LIN {X 0,Y 429.867,Z 525.018,A -85,B 0,C 180,E1 -9883.558,E2 -9883.558} C_VEL
LIN {X 0,Y 429.582,Z 537.732,A -85,B 0,C 180,E1 -9884.035,E2 -9884.035} C_VEL
LIN {X 0,Y 429.167,Z 549.996,A -85,B 0,C 180,E1 -9884.689,E2 -9884.689} C_VEL
LIN {X 0,Y 428.602,Z 561.771,A -85,B 0,C 180,E1 -9885.511,E2 -9885.511} C_VEL
LIN {X 0,Y 428.009,Z 572.562,A -85,B 0,C 180,E1 -9886.468,E2 -9886.468} C_VEL
LIN {X 0,Y 427.365,Z 583.19,A -85,B 0,C 180,E1 -9887.656,E2 -9887.656} C_VEL
LIN {X 0,Y 426.826,Z 591.861,A -85,B 0,C 180,E1 -9888.845,E2 -9888.845} C_VEL
LIN {X 0,Y 426.281,Z 598.998,A -85,B 0,C 180,E1 -9890.031,E2 -9890.031} C_VEL
LIN {X 0,Y 425.845,Z 605.937,A -85,B 0,C 180,E1 -9891.458,E2 -9891.458} C_VEL
LIN {X 0,Y 425.404,Z 611.932,A -85,B 0,C 180,E1 -9893.034,E2 -9893.034} C_VEL
LIN {X 0,Y 425.046,Z 615.71,A -85,B 0,C 180,E1 -9894.306,E2 -9894.306} C_VEL
LIN {X 0,Y 425.047,Z 617.92,A -85,B 0,C 180,E1 -9895.258,E2 -9895.258} C_VEL
LIN {X 0,Y 424.825,Z 619.716,A -85,B 0,C 180,E1 -9896.206,E2 -9896.206} C_VEL
LIN {X 0,Y 424.586,Z 621.03,A -85,B 0,C 180,E1 -9897.154,E2 -9897.154} C_VEL
LIN {X 0,Y 424.44,Z 621.926,A -85,B 0,C 180,E1 -9898.102,E2 -9898.102} C_VEL
LIN {X 0,Y 424.38,Z 622.415,A -85,B 0,C 180,E1 -9899.051,E2 -9899.051} C_VEL
LIN {X 0,Y 424.352,Z 622.464,A -85,B 0,C 180,E1 -9900,E2 -9900} C_VEL
LIN {X 0,Y 424.35,Z 622.081,A -85,B 0,C 180,E1 -9900.949,E2 -9900.949} C_VEL
LIN {X 0,Y 424.414,Z 621.294,A -85,B 0,C 180,E1 -9901.898,E2 -9901.898} C_VEL
LIN {X 0,Y 424.575,Z 620.089,A -85,B 0,C 180,E1 -9902.846,E2 -9902.846} C_VEL
LIN {X 0,Y 424.8,Z 617.445,A -85,B 0,C 180,E1 -9904.27,E2 -9904.27} C_VEL
LIN {X 0,Y 424.835,Z 613.78,A -85,B 0,C 180,E1 -9905.696,E2 -9905.696} C_VEL
LIN {X 0,Y 425.13,Z 608.245,A -85,B 0,C 180,E1 -9907.302,E2 -9907.302} C_VEL
LIN {X 0,Y 425.442,Z 601.67,A -85,B 0,C 180,E1 -9908.79,E2 -9908.79} C_VEL
LIN {X 0,Y 425.889,Z 593.769,A -85,B 0,C 180,E1 -9910.218,E2 -9910.218} C_VEL
LIN {X 0,Y 426.316,Z 585.656,A -85,B 0,C 180,E1 -9911.41,E2 -9911.41} C_VEL
LIN {X 0,Y 426.843,Z 575.754,A -85,B 0,C 180,E1 -9912.601,E2 -9912.601} C_VEL
LIN {X 0,Y 427.41,Z 564.895,A -85,B 0,C 180,E1 -9913.66,E2 -9913.66} C_VEL
LIN {X 0,Y 427.808,Z 554.016,A -85,B 0,C 180,E1 -9914.509,E2 -9914.509} C_VEL
LIN {X 0,Y 428.215,Z 541.201,A -85,B 0,C 180,E1 -9915.285,E2 -9915.285} C_VEL
LIN {X 0,Y 428.601,Z 528.47,A -85,B 0,C 180,E1 -9915.85,E2 -9915.85} C_VEL
LIN {X 0,Y 428.82,Z 515.15,A -85,B 0,C 180,E1 -9916.239,E2 -9916.239} C_VEL
LIN {X 0,Y 429.959,Z 434.183,A -85,B 0,C 180,E1 -9917.837,E2 -9917.837} C_VEL
LIN {X 0,Y 425.368,Z 420.644,A -85,B 0,C 180,E1 -9918.296,E2 -9918.296} C_VEL
LIN {X 0,Y 425.296,Z 420.514,A -85,B 0,C 180,E1 -9921.318,E2 -9921.318} C_VEL
LIN {X 0,Y 425.322,Z 420.501,A -85,B 0,C 180,E1 -9924.657,E2 -9924.657} C_VEL
LIN {X 0,Y 425.348,Z 420.498,A -85,B 0,C 180,E1 -9927.558,E2 -9927.558} C_VEL
LIN {X 0,Y 425.291,Z 420.509,A -85,B 0,C 180,E1 -9930.816,E2 -9930.816} C_VEL
LIN {X 0,Y 425.314,Z 420.49,A -85,B 0,C 180,E1 -9934.288,E2 -9934.288} C_VEL
LIN {X 0,Y 425.281,Z 420.51,A -85,B 0,C 180,E1 -9937.694,E2 -9937.694} C_VEL
LIN {X 0,Y 425.282,Z 420.5,A -85,B 0,C 180,E1 -9940.52,E2 -9940.52} C_VEL
LIN {X 0,Y 425.26,Z 420.514,A -85,B 0,C 180,E1 -9943.351,E2 -9943.351} C_VEL
LIN {X 0,Y 425.26,Z 420.506,A -85,B 0,C 180,E1 -9946.649,E2 -9946.649} C_VEL
LIN {X 0,Y 425.288,Z 420.502,A -85,B 0,C 180,E1 -9949.873,E2 -9949.873} C_VEL
LIN {X 0,Y 425.279,Z 420.511,A -85,B 0,C 180,E1 -9952.489,E2 -9952.489} C_VEL
LIN {X 0,Y 425.31,Z 420.505,A -85,B 0,C 180,E1 -9955.817,E2 -9955.817} C_VEL
LIN {X 0,Y 425.293,Z 420.511,A -85,B 0,C 180,E1 -9959.239,E2 -9959.239} C_VEL
LIN {X 0,Y 425.31,Z 420.647,A -85,B 0,C 180,E1 -9962.529,E2 -9962.529} C_VEL
LIN {X 0,Y 428.375,Z 435.146,A -85,B 0,C 180,E1 -9965.269,E2 -9965.269} C_VEL
LIN {X 0,Y 428.559,Z 439.554,A -85,B 0,C 180,E1 -9966.054,E2 -9966.054} C_VEL
LIN {X 0,Y 427.818,Z 458.202,A -85,B 0,C 180,E1 -9969.236,E2 -9969.236} C_VEL
LIN {X 0,Y 427.38,Z 471.342,A -85,B 0,C 180,E1 -9971.337,E2 -9971.337} C_VEL
LIN {X 0,Y 430.685,Z 490.935,A -85,B 0,C 180,E1 -9971.834,E2 -9971.834} C_VEL
LIN {X 0,Y 430.212,Z 535.192,A -85,B 0,C 180,E1 -9972.578,E2 -9972.578} C_VEL
LIN {X 0,Y 429.516,Z 541.034,A -85,B 0,C 180,E1 -9972.65,E2 -9972.65} C_VEL
LIN {X 0,Y 423.913,Z 560.045,A -85,B 0,C 180,E1 -9972.744,E2 -9972.744} C_VEL
LIN {X 0,Y 423.196,Z 565.888,A -85,B 0,C 180,E1 -9972.816,E2 -9972.816} C_VEL
LIN {X 0,Y 422.841,Z 583.643,A -85,B 0,C 180,E1 -9973.152,E2 -9973.152} C_VEL
LIN {X 0,Y 422.427,Z 596.784,A -85,B 0,C 180,E1 -9973.602,E2 -9973.602} C_VEL
LIN {X 0,Y 421.856,Z 609.384,A -85,B 0,C 180,E1 -9974.231,E2 -9974.231} C_VEL
LIN {X 0,Y 421.23,Z 620.994,A -85,B 0,C 180,E1 -9975.012,E2 -9975.012} C_VEL
LIN {X 0,Y 420.569,Z 632.621,A -85,B 0,C 180,E1 -9976.028,E2 -9976.028} C_VEL
LIN {X 0,Y 419.824,Z 643.18,A -85,B 0,C 180,E1 -9977.185,E2 -9977.185} C_VEL
LIN {X 0,Y 419.036,Z 652.058,A -85,B 0,C 180,E1 -9978.389,E2 -9978.389} C_VEL
LIN {X 0,Y 418.455,Z 660.712,A -85,B 0,C 180,E1 -9979.843,E2 -9979.843} C_VEL
LIN {X 0,Y 417.94,Z 667.662,A -85,B 0,C 180,E1 -9981.295,E2 -9981.295} C_VEL
LIN {X 0,Y 417.558,Z 673.185,A -85,B 0,C 180,E1 -9982.748,E2 -9982.748} C_VEL
LIN {X 0,Y 417.394,Z 677.517,A -85,B 0,C 180,E1 -9984.202,E2 -9984.202} C_VEL
LIN {X 0,Y 417.216,Z 679.799,A -85,B 0,C 180,E1 -9985.169,E2 -9985.169} C_VEL
LIN {X 0,Y 417.126,Z 681.659,A -85,B 0,C 180,E1 -9986.136,E2 -9986.136} C_VEL
LIN {X 0,Y 417.137,Z 683.08,A -85,B 0,C 180,E1 -9987.103,E2 -9987.103} C_VEL
LIN {X 0,Y 417.014,Z 684.693,A -85,B 0,C 180,E1 -9989.034,E2 -9989.034} C_VEL
LIN {X 0,Y 417.004,Z 684.929,A -85,B 0,C 180,E1 -9990,E2 -9990} C_VEL
LIN {X 0,Y 417.081,Z 684.152,A -85,B 0,C 180,E1 -9991.931,E2 -9991.931} C_VEL
LIN {X 0,Y 417.137,Z 683.186,A -85,B 0,C 180,E1 -9992.897,E2 -9992.897} C_VEL
LIN {X 0,Y 417.125,Z 681.824,A -85,B 0,C 180,E1 -9993.864,E2 -9993.864} C_VEL
LIN {X 0,Y 417.316,Z 678.955,A -85,B 0,C 180,E1 -9995.315,E2 -9995.315} C_VEL
LIN {X 0,Y 417.48,Z 675.059,A -85,B 0,C 180,E1 -9996.768,E2 -9996.768} C_VEL
LIN {X 0,Y 417.788,Z 670.009,A -85,B 0,C 180,E1 -9998.221,E2 -9998.221} C_VEL
LIN {X 0,Y 418.283,Z 663.641,A -85,B 0,C 180,E1 -9999.673,E2 -9999.673} C_VEL
LIN {X 0,Y 418.866,Z 655.73,A -85,B 0,C 180,E1 -10001.125,E2 -10001.125} C_VEL
LIN {X 0,Y 419.453,Z 647.648,A -85,B 0,C 180,E1 -10002.335,E2 -10002.335} C_VEL
LIN {X 0,Y 420.25,Z 637.715,A -85,B 0,C 180,E1 -10003.54,E2 -10003.54} C_VEL
LIN {X 0,Y 420.88,Z 626.554,A -85,B 0,C 180,E1 -10004.629,E2 -10004.629} C_VEL
LIN {X 0,Y 421.554,Z 615.626,A -85,B 0,C 180,E1 -10005.471,E2 -10005.471} C_VEL
LIN {X 0,Y 422.164,Z 604.555,A -85,B 0,C 180,E1 -10006.129,E2 -10006.129} C_VEL
LIN {X 0,Y 422.695,Z 591.407,A -85,B 0,C 180,E1 -10006.698,E2 -10006.698} C_VEL
LIN {X 0,Y 422.999,Z 579.875,A -85,B 0,C 180,E1 -10007.028,E2 -10007.028} C_VEL
LIN {X 0,Y 423.912,Z 491.011,A -85,B 0,C 180,E1 -10008.562,E2 -10008.562} C_VEL
LIN {X 0,Y 420.501,Z 471.498,A -85,B 0,C 180,E1 -10009.071,E2 -10009.071} C_VEL
LIN {X 0,Y 421.094,Z 454.836,A -85,B 0,C 180,E1 -10011.799,E2 -10011.799} C_VEL
LIN {X 0,Y 421.759,Z 438.57,A -85,B 0,C 180,E1 -10014.62,E2 -10014.62} C_VEL
LIN {X 0,Y 419.397,Z 426.486,A -85,B 0,C 180,E1 -10016.901,E2 -10016.901} C_VEL
LIN {X 0,Y 418.278,Z 421.387,A -85,B 0,C 180,E1 -10017.885,E2 -10017.885} C_VEL
LIN {X 0,Y 418.214,Z 421.393,A -85,B 0,C 180,E1 -10021.396,E2 -10021.396} C_VEL
LIN {X 0,Y 418.268,Z 421.386,A -85,B 0,C 180,E1 -10024.58,E2 -10024.58} C_VEL
LIN {X 0,Y 418.229,Z 421.388,A -85,B 0,C 180,E1 -10027.833,E2 -10027.833} C_VEL
LIN {X 0,Y 418.225,Z 421.386,A -85,B 0,C 180,E1 -10030.948,E2 -10030.948} C_VEL
LIN {X 0,Y 418.212,Z 421.385,A -85,B 0,C 180,E1 -10033.729,E2 -10033.729} C_VEL
LIN {X 0,Y 418.218,Z 421.392,A -85,B 0,C 180,E1 -10036.45,E2 -10036.45} C_VEL
LIN {X 0,Y 418.226,Z 421.387,A -85,B 0,C 180,E1 -10039.13,E2 -10039.13} C_VEL
LIN {X 0,Y 418.231,Z 421.386,A -85,B 0,C 180,E1 -10042.167,E2 -10042.167} C_VEL
LIN {X 0,Y 418.268,Z 421.381,A -85,B 0,C 180,E1 -10045.42,E2 -10045.42} C_VEL
LIN {X 0,Y 418.214,Z 421.394,A -85,B 0,C 180,E1 -10048.604,E2 -10048.604} C_VEL
LIN {X 0,Y 418.259,Z 421.386,A -85,B 0,C 180,E1 -10051.934,E2 -10051.934} C_VEL
LIN {X 0,Y 418.284,Z 421.504,A -85,B 0,C 180,E1 -10052.526,E2 -10052.526} C_VEL
LIN {X 0,Y 421.357,Z 436.857,A -85,B 0,C 180,E1 -10055.355,E2 -10055.355} C_VEL
LIN {X 0,Y 421.519,Z 441.427,A -85,B 0,C 180,E1 -10056.151,E2 -10056.151} C_VEL
LIN {X 0,Y 420.644,Z 462.332,A -85,B 0,C 180,E1 -10059.715,E2 -10059.715} C_VEL
LIN {X 0,Y 420.237,Z 471.969,A -85,B 0,C 180,E1 -10061.346,E2 -10061.346} C_VEL
LIN {X 0,Y 423.175,Z 491.893,A -85,B 0,C 180,E1 -10061.883,E2 -10061.883} C_VEL
LIN {X 0,Y 421.684,Z 582.569,A -85,B 0,C 180,E1 -10063.727,E2 -10063.727} C_VEL
LIN {X 0,Y 421.258,Z 596.208,A -85,B 0,C 180,E1 -10064.208,E2 -10064.208} C_VEL
LIN {X 0,Y 420.744,Z 609.18,A -85,B 0,C 180,E1 -10064.871,E2 -10064.871} C_VEL
LIN {X 0,Y 420.176,Z 621.079,A -85,B 0,C 180,E1 -10065.68,E2 -10065.68} C_VEL
LIN {X 0,Y 419.678,Z 632.631,A -85,B 0,C 180,E1 -10066.688,E2 -10066.688} C_VEL
LIN {X 0,Y 418.978,Z 643.706,A -85,B 0,C 180,E1 -10067.896,E2 -10067.896} C_VEL
LIN {X 0,Y 418.481,Z 652.651,A -85,B 0,C 180,E1 -10069.109,E2 -10069.109} C_VEL
LIN {X 0,Y 418.001,Z 661.355,A -85,B 0,C 180,E1 -10070.565,E2 -10070.565} C_VEL
LIN {X 0,Y 417.597,Z 668.334,A -85,B 0,C 180,E1 -10072.019,E2 -10072.019} C_VEL
LIN {X 0,Y 417.393,Z 673.725,A -85,B 0,C 180,E1 -10073.432,E2 -10073.432} C_VEL
LIN {X 0,Y 417.205,Z 678.792,A -85,B 0,C 180,E1 -10075.168,E2 -10075.168} C_VEL
LIN {X 0,Y 417.098,Z 680.906,A -85,B 0,C 180,E1 -10076.135,E2 -10076.135} C_VEL
LIN {X 0,Y 417.1,Z 682.565,A -85,B 0,C 180,E1 -10077.102,E2 -10077.102} C_VEL
LIN {X 0,Y 417.079,Z 683.807,A -85,B 0,C 180,E1 -10078.069,E2 -10078.069} C_VEL
LIN {X 0,Y 417.014,Z 684.577,A -85,B 0,C 180,E1 -10079.034,E2 -10079.034} C_VEL
LIN {X 0,Y 417.004,Z 684.936,A -85,B 0,C 180,E1 -10080,E2 -10080} C_VEL
LIN {X 0,Y 417.014,Z 684.888,A -85,B 0,C 180,E1 -10080.966,E2 -10080.966} C_VEL
LIN {X 0,Y 417.082,Z 684.371,A -85,B 0,C 180,E1 -10081.931,E2 -10081.931} C_VEL
LIN {X 0,Y 417.168,Z 683.441,A -85,B 0,C 180,E1 -10082.897,E2 -10082.897} C_VEL
LIN {X 0,Y 417.133,Z 682.105,A -85,B 0,C 180,E1 -10083.864,E2 -10083.864} C_VEL
LIN {X 0,Y 417.32,Z 679.213,A -85,B 0,C 180,E1 -10085.315,E2 -10085.315} C_VEL
LIN {X 0,Y 417.472,Z 675.228,A -85,B 0,C 180,E1 -10086.768,E2 -10086.768} C_VEL
LIN {X 0,Y 417.862,Z 669.063,A -85,B 0,C 180,E1 -10088.463,E2 -10088.463} C_VEL
LIN {X 0,Y 418.316,Z 662.293,A -85,B 0,C 180,E1 -10089.916,E2 -10089.916} C_VEL
LIN {X 0,Y 418.97,Z 653.777,A -85,B 0,C 180,E1 -10091.367,E2 -10091.367} C_VEL
LIN {X 0,Y 419.506,Z 645.109,A -85,B 0,C 180,E1 -10092.579,E2 -10092.579} C_VEL
LIN {X 0,Y 420.248,Z 634.771,A -85,B 0,C 180,E1 -10093.747,E2 -10093.747} C_VEL
LIN {X 0,Y 420.895,Z 623.794,A -85,B 0,C 180,E1 -10094.752,E2 -10094.752} C_VEL
LIN {X 0,Y 421.55,Z 612.056,A -85,B 0,C 180,E1 -10095.595,E2 -10095.595} C_VEL
LIN {X 0,Y 422.159,Z 600.099,A -85,B 0,C 180,E1 -10096.254,E2 -10096.254} C_VEL
LIN {X 0,Y 422.622,Z 587.363,A -85,B 0,C 180,E1 -10096.763,E2 -10096.763} C_VEL
LIN {X 0,Y 423.057,Z 571.747,A -85,B 0,C 180,E1 -10097.15,E2 -10097.15} C_VEL
LIN {X 0,Y 424.874,Z 497.19,A -85,B 0,C 180,E1 -10098.803,E2 -10098.803} C_VEL
LIN {X 0,Y 424.848,Z 490.529,A -85,B 0,C 180,E1 -10098.968,E2 -10098.968} C_VEL
LIN {X 0,Y 422.078,Z 475.752,A -85,B 0,C 180,E1 -10099.522,E2 -10099.522} C_VEL
LIN {X 0,Y 421.578,Z 473.354,A -85,B 0,C 180,E1 -10099.635,E2 -10099.635} C_VEL
LIN {X 0,Y 422.554,Z 453.348,A -85,B 0,C 180,E1 -10103.008,E2 -10103.008} C_VEL
LIN {X 0,Y 422.998,Z 441.224,A -85,B 0,C 180,E1 -10105.067,E2 -10105.067} C_VEL
LIN {X 0,Y 421.29,Z 432.304,A -85,B 0,C 180,E1 -10106.771,E2 -10106.771} C_VEL
LIN {X 0,Y 418.268,Z 421.389,A -85,B 0,C 180,E1 -10109.008,E2 -10109.008} C_VEL
LIN {X 0,Y 418.248,Z 421.387,A -85,B 0,C 180,E1 -10112.528,E2 -10112.528} C_VEL
LIN {X 0,Y 418.261,Z 421.385,A -85,B 0,C 180,E1 -10114.841,E2 -10114.841} C_VEL
LIN {X 0,Y 418.257,Z 421.384,A -85,B 0,C 180,E1 -10118.442,E2 -10118.442} C_VEL
LIN {X 0,Y 418.224,Z 421.39,A -85,B 0,C 180,E1 -10120.948,E2 -10120.948} C_VEL
LIN {X 0,Y 418.212,Z 421.391,A -85,B 0,C 180,E1 -10123.729,E2 -10123.729} C_VEL
LIN {X 0,Y 418.212,Z 421.393,A -85,B 0,C 180,E1 -10126.449,E2 -10126.449} C_VEL
LIN {X 0,Y 418.226,Z 421.388,A -85,B 0,C 180,E1 -10129.13,E2 -10129.13} C_VEL
LIN {X 0,Y 418.229,Z 421.388,A -85,B 0,C 180,E1 -10132.167,E2 -10132.167} C_VEL
LIN {X 0,Y 418.267,Z 421.383,A -85,B 0,C 180,E1 -10135.42,E2 -10135.42} C_VEL
LIN {X 0,Y 418.213,Z 421.393,A -85,B 0,C 180,E1 -10138.604,E2 -10138.604} C_VEL
LIN {X 0,Y 418.297,Z 421.512,A -85,B 0,C 180,E1 -10139.671,E2 -10139.671} C_VEL
LIN {X 0,Y 421.825,Z 438.127,A -85,B 0,C 180,E1 -10142.73,E2 -10142.73} C_VEL
LIN {X 0,Y 422.231,Z 441.312,A -85,B 0,C 180,E1 -10143.294,E2 -10143.294} C_VEL
LIN {X 0,Y 421.27,Z 456.799,A -85,B 0,C 180,E1 -10145.875,E2 -10145.875} C_VEL
LIN {X 0,Y 420.182,Z 475.297,A -85,B 0,C 180,E1 -10148.924,E2 -10148.924} C_VEL
LIN {X 0,Y 419.678,Z 485.648,A -85,B 0,C 180,E1 -10150.591,E2 -10150.591} C_VEL
LIN {X 0,Y 421.506,Z 499.502,A -85,B 0,C 180,E1 -10151.079,E2 -10151.079} C_VEL
LIN {X 0,Y 423.449,Z 519.644,A -85,B 0,C 180,E1 -10151.71,E2 -10151.71} C_VEL
LIN {X 0,Y 422.991,Z 539.758,A -85,B 0,C 180,E1 -10152.153,E2 -10152.153} C_VEL
LIN {X 0,Y 422.267,Z 602.397,A -85,B 0,C 180,E1 -10153.222,E2 -10153.222} C_VEL
LIN {X 0,Y 421.922,Z 615.066,A -85,B 0,C 180,E1 -10153.581,E2 -10153.581} C_VEL
LIN {X 0,Y 421.352,Z 627.88,A -85,B 0,C 180,E1 -10154.149,E2 -10154.149} C_VEL
LIN {X 0,Y 420.681,Z 639.693,A -85,B 0,C 180,E1 -10154.868,E2 -10154.868} C_VEL
LIN {X 0,Y 420.07,Z 650.411,A -85,B 0,C 180,E1 -10155.713,E2 -10155.713} C_VEL
LIN {X 0,Y 419.343,Z 661.316,A -85,B 0,C 180,E1 -10156.8,E2 -10156.8} C_VEL
LIN {X 0,Y 418.764,Z 670.173,A -85,B 0,C 180,E1 -10157.89,E2 -10157.89} C_VEL
LIN {X 0,Y 418.228,Z 678.289,A -85,B 0,C 180,E1 -10159.103,E2 -10159.103} C_VEL
LIN {X 0,Y 417.746,Z 686.236,A -85,B 0,C 180,E1 -10160.559,E2 -10160.559} C_VEL
LIN {X 0,Y 417.464,Z 691.604,A -85,B 0,C 180,E1 -10161.773,E2 -10161.773} C_VEL
LIN {X 0,Y 417.236,Z 696.843,A -85,B 0,C 180,E1 -10163.229,E2 -10163.229} C_VEL
LIN {X 0,Y 417.159,Z 700.89,A -85,B 0,C 180,E1 -10164.683,E2 -10164.683} C_VEL
LIN {X 0,Y 417.095,Z 703.869,A -85,B 0,C 180,E1 -10166.135,E2 -10166.135} C_VEL
LIN {X 0,Y 417.116,Z 705.313,A -85,B 0,C 180,E1 -10167.103,E2 -10167.103} C_VEL
LIN {X 0,Y 417.097,Z 706.349,A -85,B 0,C 180,E1 -10168.069,E2 -10168.069} C_VEL
LIN {X 0,Y 417.063,Z 706.954,A -85,B 0,C 180,E1 -10169.034,E2 -10169.034} C_VEL
LIN {X 0,Y 417.066,Z 707.145,A -85,B 0,C 180,E1 -10170,E2 -10170} C_VEL
LIN {X 0,Y 417.063,Z 706.923,A -85,B 0,C 180,E1 -10170.966,E2 -10170.966} C_VEL
LIN {X 0,Y 417.1,Z 706.307,A -85,B 0,C 180,E1 -10171.931,E2 -10171.931} C_VEL
LIN {X 0,Y 417.12,Z 705.298,A -85,B 0,C 180,E1 -10172.897,E2 -10172.897} C_VEL
LIN {X 0,Y 417.103,Z 703.864,A -85,B 0,C 180,E1 -10173.865,E2 -10173.865} C_VEL
LIN {X 0,Y 417.161,Z 700.881,A -85,B 0,C 180,E1 -10175.317,E2 -10175.317} C_VEL
LIN {X 0,Y 417.265,Z 696.83,A -85,B 0,C 180,E1 -10176.771,E2 -10176.771} C_VEL
LIN {X 0,Y 417.523,Z 690.581,A -85,B 0,C 180,E1 -10178.47,E2 -10178.47} C_VEL
LIN {X 0,Y 417.892,Z 683.761,A -85,B 0,C 180,E1 -10179.926,E2 -10179.926} C_VEL
LIN {X 0,Y 418.34,Z 676.779,A -85,B 0,C 180,E1 -10181.139,E2 -10181.139} C_VEL
LIN {X 0,Y 418.915,Z 668.339,A -85,B 0,C 180,E1 -10182.351,E2 -10182.351} C_VEL
LIN {X 0,Y 419.61,Z 657.886,A -85,B 0,C 180,E1 -10183.561,E2 -10183.561} C_VEL
LIN {X 0,Y 420.216,Z 647.518,A -85,B 0,C 180,E1 -10184.529,E2 -10184.529} C_VEL
LIN {X 0,Y 420.91,Z 636.08,A -85,B 0,C 180,E1 -10185.371,E2 -10185.371} C_VEL
LIN {X 0,Y 421.565,Z 624.189,A -85,B 0,C 180,E1 -10186.029,E2 -10186.029} C_VEL
LIN {X 0,Y 422.051,Z 611.321,A -85,B 0,C 180,E1 -10186.538,E2 -10186.538} C_VEL
LIN {X 0,Y 422.393,Z 599.213,A -85,B 0,C 180,E1 -10186.835,E2 -10186.835} C_VEL
LIN {X 0,Y 424.12,Z 518.65,A -85,B 0,C 180,E1 -10188.602,E2 -10188.602} C_VEL
LIN {X 0,Y 421.861,Z 496.233,A -85,B 0,C 180,E1 -10189.288,E2 -10189.288} C_VEL
LIN {X 0,Y 419.734,Z 482.953,A -85,B 0,C 180,E1 -10189.775,E2 -10189.775} C_VEL
LIN {X 0,Y 421.144,Z 461.891,A -85,B 0,C 180,E1 -10193.388,E2 -10193.388} C_VEL
LIN {X 0,Y 422.78,Z 442.084,A -85,B 0,C 180,E1 -10196.935,E2 -10196.935} C_VEL
LIN {X 0,Y 421.389,Z 433.82,A -85,B 0,C 180,E1 -10198.657,E2 -10198.657} C_VEL
LIN {X 0,Y 418.708,Z 423.163,A -85,B 0,C 180,E1 -10201.126,E2 -10201.126} C_VEL
LIN {X 0,Y 418.247,Z 421.391,A -85,B 0,C 180,E1 -10201.605,E2 -10201.605} C_VEL
LIN {X 0,Y 418.261,Z 421.387,A -85,B 0,C 180,E1 -10204.841,E2 -10204.841} C_VEL
LIN {X 0,Y 418.249,Z 421.386,A -85,B 0,C 180,E1 -10208.442,E2 -10208.442} C_VEL
LIN {X 0,Y 418.221,Z 421.39,A -85,B 0,C 180,E1 -10210.948,E2 -10210.948} C_VEL
LIN {X 0,Y 418.211,Z 421.391,A -85,B 0,C 180,E1 -10213.729,E2 -10213.729} C_VEL
LIN {X 0,Y 418.211,Z 421.391,A -85,B 0,C 180,E1 -10216.449,E2 -10216.449} C_VEL
LIN {X 0,Y 418.226,Z 421.392,A -85,B 0,C 180,E1 -10219.13,E2 -10219.13} C_VEL
LIN {X 0,Y 418.231,Z 421.387,A -85,B 0,C 180,E1 -10222.167,E2 -10222.167} C_VEL
LIN {X 0,Y 418.268,Z 421.383,A -85,B 0,C 180,E1 -10225.42,E2 -10225.42} C_VEL
LIN {X 0,Y 418.214,Z 421.392,A -85,B 0,C 180,E1 -10228.604,E2 -10228.604} C_VEL
LIN {X 0,Y 418.294,Z 421.382,A -85,B 0,C 180,E1 -10231.937,E2 -10231.937} C_VEL
LIN {X 0,Y 418.292,Z 421.385,A -85,B 0,C 180,E1 -10235.163,E2 -10235.163} C_VEL
LIN {X 0,Y 418.237,Z 421.392,A -85,B 0,C 180,E1 -10238.304,E2 -10238.304} C_VEL
LIN {X 0,Y 418.286,Z 421.384,A -85,B 0,C 180,E1 -10240.269,E2 -10240.269} C_VEL
LIN {X 0,Y 419.333,Z 424.277,A -85,B 0,C 180,E1 -10240.431,E2 -10240.431} C_VEL
LIN {X 0,Y 424.852,Z 436.499,A -85,B 0,C 180,E1 -10241.141,E2 -10241.141} C_VEL
LIN {X 0,Y 425.474,Z 438.692,A -85,B 0,C 180,E1 -10241.237,E2 -10241.237} C_VEL
LIN {X 0,Y 423.251,Z 524.575,A -85,B 0,C 180,E1 -10243.2,E2 -10243.2} C_VEL
LIN {X 0,Y 422.931,Z 537.536,A -85,B 0,C 180,E1 -10243.684,E2 -10243.684} C_VEL
LIN {X 0,Y 422.527,Z 549.641,A -85,B 0,C 180,E1 -10244.318,E2 -10244.318} C_VEL
LIN {X 0,Y 421.919,Z 562.009,A -85,B 0,C 180,E1 -10245.182,E2 -10245.182} C_VEL
LIN {X 0,Y 421.291,Z 572.639,A -85,B 0,C 180,E1 -10246.125,E2 -10246.125} C_VEL
LIN {X 0,Y 420.681,Z 582.463,A -85,B 0,C 180,E1 -10247.211,E2 -10247.211} C_VEL
LIN {X 0,Y 420.057,Z 591.348,A -85,B 0,C 180,E1 -10248.418,E2 -10248.418} C_VEL
LIN {X 0,Y 419.364,Z 600.004,A -85,B 0,C 180,E1 -10249.865,E2 -10249.865} C_VEL
LIN {X 0,Y 418.892,Z 606.865,A -85,B 0,C 180,E1 -10251.315,E2 -10251.315} C_VEL
LIN {X 0,Y 418.421,Z 612.841,A -85,B 0,C 180,E1 -10252.919,E2 -10252.919} C_VEL
LIN {X 0,Y 418.032,Z 616.579,A -85,B 0,C 180,E1 -10254.211,E2 -10254.211} C_VEL
LIN {X 0,Y 418.026,Z 618.772,A -85,B 0,C 180,E1 -10255.178,E2 -10255.178} C_VEL
LIN {X 0,Y 417.796,Z 620.534,A -85,B 0,C 180,E1 -10256.142,E2 -10256.142} C_VEL
LIN {X 0,Y 417.545,Z 621.824,A -85,B 0,C 180,E1 -10257.106,E2 -10257.106} C_VEL
LIN {X 0,Y 417.387,Z 622.698,A -85,B 0,C 180,E1 -10258.07,E2 -10258.07} C_VEL
LIN {X 0,Y 417.321,Z 623.158,A -85,B 0,C 180,E1 -10259.035,E2 -10259.035} C_VEL
LIN {X 0,Y 417.287,Z 623.161,A -85,B 0,C 180,E1 -10260,E2 -10260} C_VEL
LIN {X 0,Y 417.29,Z 622.749,A -85,B 0,C 180,E1 -10260.965,E2 -10260.965} C_VEL
LIN {X 0,Y 417.362,Z 621.931,A -85,B 0,C 180,E1 -10261.93,E2 -10261.93} C_VEL
LIN {X 0,Y 417.533,Z 620.679,A -85,B 0,C 180,E1 -10262.895,E2 -10262.895} C_VEL
LIN {X 0,Y 417.737,Z 617.983,A -85,B 0,C 180,E1 -10264.342,E2 -10264.342} C_VEL
LIN {X 0,Y 417.775,Z 614.253,A -85,B 0,C 180,E1 -10265.793,E2 -10265.793} C_VEL
LIN {X 0,Y 418.095,Z 608.908,A -85,B 0,C 180,E1 -10267.356,E2 -10267.356} C_VEL
LIN {X 0,Y 418.42,Z 601.988,A -85,B 0,C 180,E1 -10268.938,E2 -10268.938} C_VEL
LIN {X 0,Y 418.881,Z 593.966,A -85,B 0,C 180,E1 -10270.391,E2 -10270.391} C_VEL
LIN {X 0,Y 419.461,Z 583.915,A -85,B 0,C 180,E1 -10271.844,E2 -10271.844} C_VEL
LIN {X 0,Y 420.021,Z 573.444,A -85,B 0,C 180,E1 -10273.055,E2 -10273.055} C_VEL
LIN {X 0,Y 420.609,Z 561.403,A -85,B 0,C 180,E1 -10274.164,E2 -10274.164} C_VEL
LIN {X 0,Y 421.045,Z 549.947,A -85,B 0,C 180,E1 -10274.994,E2 -10274.994} C_VEL
LIN {X 0,Y 421.445,Z 537.954,A -85,B 0,C 180,E1 -10275.661,E2 -10275.661} C_VEL
LIN {X 0,Y 421.816,Z 524.384,A -85,B 0,C 180,E1 -10276.205,E2 -10276.205} C_VEL
LIN {X 0,Y 421.989,Z 509.448,A -85,B 0,C 180,E1 -10276.571,E2 -10276.571} C_VEL
LIN {X 0,Y 423.228,Z 436.539,A -85,B 0,C 180,E1 -10278.039,E2 -10278.039} C_VEL
LIN {X 0,Y 418.339,Z 421.378,A -85,B 0,C 180,E1 -10278.578,E2 -10278.578} C_VEL
LIN {X 0,Y 418.237,Z 421.387,A -85,B 0,C 180,E1 -10281.696,E2 -10281.696} C_VEL
LIN {X 0,Y 418.287,Z 421.379,A -85,B 0,C 180,E1 -10284.864,E2 -10284.864} C_VEL
LIN {X 0,Y 418.292,Z 421.375,A -85,B 0,C 180,E1 -10288.063,E2 -10288.063} C_VEL
LIN {X 0,Y 418.214,Z 421.385,A -85,B 0,C 180,E1 -10291.396,E2 -10291.396} C_VEL
LIN {X 0,Y 418.268,Z 421.368,A -85,B 0,C 180,E1 -10294.58,E2 -10294.58} C_VEL
LIN {X 0,Y 418.23,Z 421.388,A -85,B 0,C 180,E1 -10297.833,E2 -10297.833} C_VEL
LIN {X 0,Y 418.224,Z 421.38,A -85,B 0,C 180,E1 -10300.948,E2 -10300.948} C_VEL
LIN {X 0,Y 418.212,Z 421.39,A -85,B 0,C 180,E1 -10303.729,E2 -10303.729} C_VEL
LIN {X 0,Y 418.211,Z 421.382,A -85,B 0,C 180,E1 -10306.449,E2 -10306.449} C_VEL
LIN {X 0,Y 418.225,Z 421.384,A -85,B 0,C 180,E1 -10309.13,E2 -10309.13} C_VEL
LIN {X 0,Y 418.229,Z 421.39,A -85,B 0,C 180,E1 -10312.167,E2 -10312.167} C_VEL
LIN {X 0,Y 418.268,Z 421.381,A -85,B 0,C 180,E1 -10315.42,E2 -10315.42} C_VEL
LIN {X 0,Y 418.214,Z 421.393,A -85,B 0,C 180,E1 -10318.604,E2 -10318.604} C_VEL
LIN {X 0,Y 418.25,Z 421.393,A -85,B 0,C 180,E1 -10321.934,E2 -10321.934} C_VEL
LIN {X 0,Y 418.249,Z 421.459,A -85,B 0,C 180,E1 -10322.241,E2 -10322.241} C_VEL
LIN {X 0,Y 421.473,Z 436.584,A -85,B 0,C 180,E1 -10325.128,E2 -10325.128} C_VEL
LIN {X 0,Y 421.691,Z 440.869,A -85,B 0,C 180,E1 -10325.9,E2 -10325.9} C_VEL
LIN {X 0,Y 420.88,Z 460.409,A -85,B 0,C 180,E1 -10329.246,E2 -10329.246} C_VEL
LIN {X 0,Y 420.491,Z 471.478,A -85,B 0,C 180,E1 -10331.023,E2 -10331.023} C_VEL
LIN {X 0,Y 423.94,Z 491.511,A -85,B 0,C 180,E1 -10331.543,E2 -10331.543} C_VEL
LIN {X 0,Y 423.196,Z 565.888,A -85,B 0,C 180,E1 -10332.816,E2 -10332.816} C_VEL
LIN {X 0,Y 422.457,Z 571.734,A -85,B 0,C 180,E1 -10332.887,E2 -10332.887} C_VEL
LIN {X 0,Y 419.537,Z 581.213,A -85,B 0,C 180,E1 -10332.955,E2 -10332.955} C_VEL
LIN {X 0,Y 416.566,Z 590.577,A -85,B 0,C 180,E1 -10333.106,E2 -10333.106} C_VEL
LIN {X 0,Y 415.714,Z 596.234,A -85,B 0,C 180,E1 -10333.297,E2 -10333.297} C_VEL
LIN {X 0,Y 415.103,Z 608.488,A -85,B 0,C 180,E1 -10333.904,E2 -10333.904} C_VEL
LIN {X 0,Y 414.482,Z 619.563,A -85,B 0,C 180,E1 -10334.637,E2 -10334.637} C_VEL
LIN {X 0,Y 413.795,Z 630.751,A -85,B 0,C 180,E1 -10335.588,E2 -10335.588} C_VEL
LIN {X 0,Y 413.073,Z 641.318,A -85,B 0,C 180,E1 -10336.721,E2 -10336.721} C_VEL
LIN {X 0,Y 412.258,Z 650.617,A -85,B 0,C 180,E1 -10337.946,E2 -10337.946} C_VEL
LIN {X 0,Y 411.565,Z 659.581,A -85,B 0,C 180,E1 -10339.422,E2 -10339.422} C_VEL
LIN {X 0,Y 410.996,Z 666.773,A -85,B 0,C 180,E1 -10340.899,E2 -10340.899} C_VEL
LIN {X 0,Y 410.514,Z 673.374,A -85,B 0,C 180,E1 -10342.623,E2 -10342.623} C_VEL
LIN {X 0,Y 410.33,Z 677.706,A -85,B 0,C 180,E1 -10344.101,E2 -10344.101} C_VEL
LIN {X 0,Y 410.159,Z 679.988,A -85,B 0,C 180,E1 -10345.085,E2 -10345.085} C_VEL
LIN {X 0,Y 410.039,Z 681.849,A -85,B 0,C 180,E1 -10346.069,E2 -10346.069} C_VEL
LIN {X 0,Y 410.04,Z 683.269,A -85,B 0,C 180,E1 -10347.053,E2 -10347.053} C_VEL
LIN {X 0,Y 410.012,Z 684.265,A -85,B 0,C 180,E1 -10348.035,E2 -10348.035} C_VEL
LIN {X 0,Y 409.927,Z 685.117,A -85,B 0,C 180,E1 -10350,E2 -10350} C_VEL
LIN {X 0,Y 410.012,Z 684.34,A -85,B 0,C 180,E1 -10351.965,E2 -10351.965} C_VEL
LIN {X 0,Y 410.039,Z 683.374,A -85,B 0,C 180,E1 -10352.947,E2 -10352.947} C_VEL
LIN {X 0,Y 410.038,Z 682.012,A -85,B 0,C 180,E1 -10353.931,E2 -10353.931} C_VEL
LIN {X 0,Y 410.262,Z 679.141,A -85,B 0,C 180,E1 -10355.406,E2 -10355.406} C_VEL
LIN {X 0,Y 410.429,Z 675.245,A -85,B 0,C 180,E1 -10356.884,E2 -10356.884} C_VEL
LIN {X 0,Y 410.756,Z 670.194,A -85,B 0,C 180,E1 -10358.362,E2 -10358.362} C_VEL
LIN {X 0,Y 411.276,Z 663.824,A -85,B 0,C 180,E1 -10359.839,E2 -10359.839} C_VEL
LIN {X 0,Y 411.891,Z 655.912,A -85,B 0,C 180,E1 -10361.316,E2 -10361.316} C_VEL
LIN {X 0,Y 412.531,Z 647.826,A -85,B 0,C 180,E1 -10362.545,E2 -10362.545} C_VEL
LIN {X 0,Y 413.342,Z 637.889,A -85,B 0,C 180,E1 -10363.771,E2 -10363.771} C_VEL
LIN {X 0,Y 414.023,Z 626.723,A -85,B 0,C 180,E1 -10364.877,E2 -10364.877} C_VEL
LIN {X 0,Y 414.708,Z 615.788,A -85,B 0,C 180,E1 -10365.733,E2 -10365.733} C_VEL
LIN {X 0,Y 415.357,Z 604.703,A -85,B 0,C 180,E1 -10366.401,E2 -10366.401} C_VEL
LIN {X 0,Y 415.896,Z 591.533,A -85,B 0,C 180,E1 -10366.979,E2 -10366.979} C_VEL
LIN {X 0,Y 416.216,Z 579.958,A -85,B 0,C 180,E1 -10367.314,E2 -10367.314} C_VEL
LIN {X 0,Y 417.218,Z 491.962,A -85,B 0,C 180,E1 -10368.855,E2 -10368.855} C_VEL
LIN {X 0,Y 413.663,Z 471.53,A -85,B 0,C 180,E1 -10369.413,E2 -10369.413} C_VEL
LIN {X 0,Y 414.277,Z 454.824,A -85,B 0,C 180,E1 -10372.177,E2 -10372.177} C_VEL
LIN {X 0,Y 414.903,Z 441.333,A -85,B 0,C 180,E1 -10374.52,E2 -10374.52} C_VEL
LIN {X 0,Y 414.041,Z 435.42,A -85,B 0,C 180,E1 -10375.642,E2 -10375.642} C_VEL
LIN {X 0,Y 411.213,Z 422.265,A -85,B 0,C 180,E1 -10378.208,E2 -10378.208} C_VEL
LIN {X 0,Y 411.185,Z 422.268,A -85,B 0,C 180,E1 -10381.284,E2 -10381.284} C_VEL
LIN {X 0,Y 411.208,Z 422.265,A -85,B 0,C 180,E1 -10384.334,E2 -10384.334} C_VEL
LIN {X 0,Y 411.195,Z 422.264,A -85,B 0,C 180,E1 -10387.974,E2 -10387.974} C_VEL
LIN {X 0,Y 411.166,Z 422.269,A -85,B 0,C 180,E1 -10391.228,E2 -10391.228} C_VEL
LIN {X 0,Y 411.18,Z 422.262,A -85,B 0,C 180,E1 -10394.49,E2 -10394.49} C_VEL
LIN {X 0,Y 411.181,Z 422.259,A -85,B 0,C 180,E1 -10398.195,E2 -10398.195} C_VEL
LIN {X 0,Y 411.222,Z 422.266,A -85,B 0,C 180,E1 -10400.776,E2 -10400.776} C_VEL
LIN {X 0,Y 411.2,Z 422.255,A -85,B 0,C 180,E1 -10404.471,E2 -10404.471} C_VEL
LIN {X 0,Y 411.21,Z 422.265,A -85,B 0,C 180,E1 -10406.873,E2 -10406.873} C_VEL
LIN {X 0,Y 411.213,Z 422.265,A -85,B 0,C 180,E1 -10410.65,E2 -10410.65} C_VEL
LIN {X 0,Y 411.25,Z 422.439,A -85,B 0,C 180,E1 -10412.314,E2 -10412.314} C_VEL
LIN {X 0,Y 414.115,Z 436.278,A -85,B 0,C 180,E1 -10414.895,E2 -10414.895} C_VEL
LIN {X 0,Y 414.64,Z 440.912,A -85,B 0,C 180,E1 -10415.73,E2 -10415.73} C_VEL
LIN {X 0,Y 413.809,Z 459.027,A -85,B 0,C 180,E1 -10418.844,E2 -10418.844} C_VEL
LIN {X 0,Y 413.301,Z 472.115,A -85,B 0,C 180,E1 -10421.086,E2 -10421.086} C_VEL
LIN {X 0,Y 416.298,Z 492.651,A -85,B 0,C 180,E1 -10421.649,E2 -10421.649} C_VEL
LIN {X 0,Y 414.734,Z 583.118,A -85,B 0,C 180,E1 -10423.542,E2 -10423.542} C_VEL
LIN {X 0,Y 414.28,Z 597.317,A -85,B 0,C 180,E1 -10424.061,E2 -10424.061} C_VEL
LIN {X 0,Y 413.747,Z 609.978,A -85,B 0,C 180,E1 -10424.735,E2 -10424.735} C_VEL
LIN {X 0,Y 413.158,Z 622.049,A -85,B 0,C 180,E1 -10425.581,E2 -10425.581} C_VEL
LIN {X 0,Y 412.651,Z 633.194,A -85,B 0,C 180,E1 -10426.582,E2 -10426.582} C_VEL
LIN {X 0,Y 412.033,Z 643.197,A -85,B 0,C 180,E1 -10427.689,E2 -10427.689} C_VEL
LIN {X 0,Y 411.475,Z 652.307,A -85,B 0,C 180,E1 -10428.922,E2 -10428.922} C_VEL
LIN {X 0,Y 410.953,Z 661.109,A -85,B 0,C 180,E1 -10430.401,E2 -10430.401} C_VEL
LIN {X 0,Y 410.543,Z 668.203,A -85,B 0,C 180,E1 -10431.881,E2 -10431.881} C_VEL
LIN {X 0,Y 410.311,Z 674.072,A -85,B 0,C 180,E1 -10433.441,E2 -10433.441} C_VEL
LIN {X 0,Y 410.143,Z 678.802,A -85,B 0,C 180,E1 -10435.085,E2 -10435.085} C_VEL
LIN {X 0,Y 410.013,Z 680.971,A -85,B 0,C 180,E1 -10436.068,E2 -10436.068} C_VEL
LIN {X 0,Y 410,Z 682.657,A -85,B 0,C 180,E1 -10437.052,E2 -10437.052} C_VEL
LIN {X 0,Y 410.008,Z 683.931,A -85,B 0,C 180,E1 -10438.035,E2 -10438.035} C_VEL
LIN {X 0,Y 409.939,Z 684.742,A -85,B 0,C 180,E1 -10439.018,E2 -10439.018} C_VEL
LIN {X 0,Y 409.927,Z 685.124,A -85,B 0,C 180,E1 -10440,E2 -10440} C_VEL
LIN {X 0,Y 409.939,Z 685.101,A -85,B 0,C 180,E1 -10440.982,E2 -10440.982} C_VEL
LIN {X 0,Y 410.013,Z 684.618,A -85,B 0,C 180,E1 -10441.965,E2 -10441.965} C_VEL
LIN {X 0,Y 410.085,Z 683.706,A -85,B 0,C 180,E1 -10442.947,E2 -10442.947} C_VEL
LIN {X 0,Y 410.046,Z 682.393,A -85,B 0,C 180,E1 -10443.931,E2 -10443.931} C_VEL
LIN {X 0,Y 410.274,Z 679.54,A -85,B 0,C 180,E1 -10445.406,E2 -10445.406} C_VEL
LIN {X 0,Y 410.427,Z 675.602,A -85,B 0,C 180,E1 -10446.884,E2 -10446.884} C_VEL
LIN {X 0,Y 410.777,Z 670.448,A -85,B 0,C 180,E1 -10448.362,E2 -10448.362} C_VEL
LIN {X 0,Y 411.252,Z 663.97,A -85,B 0,C 180,E1 -10449.84,E2 -10449.84} C_VEL
LIN {X 0,Y 411.904,Z 655.888,A -85,B 0,C 180,E1 -10451.316,E2 -10451.316} C_VEL
LIN {X 0,Y 412.496,Z 647.57,A -85,B 0,C 180,E1 -10452.546,E2 -10452.546} C_VEL
LIN {X 0,Y 413.254,Z 637.424,A -85,B 0,C 180,E1 -10453.774,E2 -10453.774} C_VEL
LIN {X 0,Y 414.022,Z 625.999,A -85,B 0,C 180,E1 -10454.877,E2 -10454.877} C_VEL
LIN {X 0,Y 414.64,Z 614.851,A -85,B 0,C 180,E1 -10455.735,E2 -10455.735} C_VEL
LIN {X 0,Y 415.342,Z 602.554,A -85,B 0,C 180,E1 -10456.465,E2 -10456.465} C_VEL
LIN {X 0,Y 415.931,Z 589.294,A -85,B 0,C 180,E1 -10457.041,E2 -10457.041} C_VEL
LIN {X 0,Y 416.401,Z 575.022,A -85,B 0,C 180,E1 -10457.433,E2 -10457.433} C_VEL
LIN {X 0,Y 418.435,Z 497.676,A -85,B 0,C 180,E1 -10459.198,E2 -10459.198} C_VEL
LIN {X 0,Y 418.353,Z 490.916,A -85,B 0,C 180,E1 -10459.382,E2 -10459.382} C_VEL
LIN {X 0,Y 415.433,Z 475.804,A -85,B 0,C 180,E1 -10459.99,E2 -10459.99} C_VEL
LIN {X 0,Y 414.951,Z 473.459,A -85,B 0,C 180,E1 -10460.123,E2 -10460.123} C_VEL
LIN {X 0,Y 416.091,Z 452.855,A -85,B 0,C 180,E1 -10463.65,E2 -10463.65} C_VEL
LIN {X 0,Y 416.423,Z 443.697,A -85,B 0,C 180,E1 -10465.223,E2 -10465.223} C_VEL
LIN {X 0,Y 414.75,Z 434.793,A -85,B 0,C 180,E1 -10466.954,E2 -10466.954} C_VEL
LIN {X 0,Y 412.021,Z 424.921,A -85,B 0,C 180,E1 -10469.009,E2 -10469.009} C_VEL
LIN {X 0,Y 411.205,Z 422.27,A -85,B 0,C 180,E1 -10469.598,E2 -10469.598} C_VEL
LIN {X 0,Y 411.209,Z 422.267,A -85,B 0,C 180,E1 -10473.156,E2 -10473.156} C_VEL
LIN {X 0,Y 411.194,Z 422.263,A -85,B 0,C 180,E1 -10476.552,E2 -10476.552} C_VEL
LIN {X 0,Y 411.215,Z 422.261,A -85,B 0,C 180,E1 -10479.728,E2 -10479.728} C_VEL
LIN {X 0,Y 411.176,Z 422.266,A -85,B 0,C 180,E1 -10483.133,E2 -10483.133} C_VEL
LIN {X 0,Y 411.17,Z 422.268,A -85,B 0,C 180,E1 -10485.881,E2 -10485.881} C_VEL
LIN {X 0,Y 411.166,Z 422.267,A -85,B 0,C 180,E1 -10488.772,E2 -10488.772} C_VEL
LIN {X 0,Y 411.206,Z 422.262,A -85,B 0,C 180,E1 -10491.831,E2 -10491.831} C_VEL
LIN {X 0,Y 411.212,Z 422.264,A -85,B 0,C 180,E1 -10495.122,E2 -10495.122} C_VEL
LIN {X 0,Y 411.168,Z 422.267,A -85,B 0,C 180,E1 -10498.003,E2 -10498.003} C_VEL
LIN {X 0,Y 411.246,Z 422.388,A -85,B 0,C 180,E1 -10499.442,E2 -10499.442} C_VEL
LIN {X 0,Y 414.756,Z 438.963,A -85,B 0,C 180,E1 -10502.543,E2 -10502.543} C_VEL
LIN {X 0,Y 415.271,Z 442.084,A -85,B 0,C 180,E1 -10503.109,E2 -10503.109} C_VEL
LIN {X 0,Y 414.293,Z 457.442,A -85,B 0,C 180,E1 -10505.709,E2 -10505.709} C_VEL
LIN {X 0,Y 413.312,Z 474.389,A -85,B 0,C 180,E1 -10508.556,E2 -10508.556} C_VEL
LIN {X 0,Y 412.777,Z 483.043,A -85,B 0,C 180,E1 -10509.997,E2 -10509.997} C_VEL
LIN {X 0,Y 415.029,Z 498.91,A -85,B 0,C 180,E1 -10510.629,E2 -10510.629} C_VEL
LIN {X 0,Y 416.968,Z 520.948,A -85,B 0,C 180,E1 -10511.341,E2 -10511.341} C_VEL
LIN {X 0,Y 416.129,Z 551.917,A -85,B 0,C 180,E1 -10512.064,E2 -10512.064} C_VEL
LIN {X 0,Y 415.459,Z 603.778,A -85,B 0,C 180,E1 -10512.971,E2 -10512.971} C_VEL
LIN {X 0,Y 415.052,Z 616.492,A -85,B 0,C 180,E1 -10513.365,E2 -10513.365} C_VEL
LIN {X 0,Y 414.422,Z 629.964,A -85,B 0,C 180,E1 -10514.004,E2 -10514.004} C_VEL
LIN {X 0,Y 413.722,Z 641.26,A -85,B 0,C 180,E1 -10514.734,E2 -10514.734} C_VEL
LIN {X 0,Y 413.02,Z 652.865,A -85,B 0,C 180,E1 -10515.716,E2 -10515.716} C_VEL
LIN {X 0,Y 412.22,Z 663.27,A -85,B 0,C 180,E1 -10516.819,E2 -10516.819} C_VEL
LIN {X 0,Y 411.704,Z 671.771,A -85,B 0,C 180,E1 -10517.93,E2 -10517.93} C_VEL
LIN {X 0,Y 411.085,Z 679.58,A -85,B 0,C 180,E1 -10519.16,E2 -10519.16} C_VEL
LIN {X 0,Y 410.63,Z 687.184,A -85,B 0,C 180,E1 -10520.642,E2 -10520.642} C_VEL
LIN {X 0,Y 410.3,Z 693.287,A -85,B 0,C 180,E1 -10522.124,E2 -10522.124} C_VEL
LIN {X 0,Y 410.101,Z 698.385,A -85,B 0,C 180,E1 -10523.701,E2 -10523.701} C_VEL
LIN {X 0,Y 410.077,Z 701.787,A -85,B 0,C 180,E1 -10525.084,E2 -10525.084} C_VEL
LIN {X 0,Y 410.008,Z 703.677,A -85,B 0,C 180,E1 -10526.068,E2 -10526.068} C_VEL
LIN {X 0,Y 410.013,Z 705.141,A -85,B 0,C 180,E1 -10527.052,E2 -10527.052} C_VEL
LIN {X 0,Y 410.025,Z 706.178,A -85,B 0,C 180,E1 -10528.035,E2 -10528.035} C_VEL
LIN {X 0,Y 409.985,Z 706.773,A -85,B 0,C 180,E1 -10529.018,E2 -10529.018} C_VEL
LIN {X 0,Y 409.985,Z 706.957,A -85,B 0,C 180,E1 -10530,E2 -10530} C_VEL
LIN {X 0,Y 409.985,Z 706.735,A -85,B 0,C 180,E1 -10530.982,E2 -10530.982} C_VEL
LIN {X 0,Y 410.028,Z 706.118,A -85,B 0,C 180,E1 -10531.965,E2 -10531.965} C_VEL
LIN {X 0,Y 410.018,Z 705.108,A -85,B 0,C 180,E1 -10532.948,E2 -10532.948} C_VEL
LIN {X 0,Y 410.016,Z 703.674,A -85,B 0,C 180,E1 -10533.931,E2 -10533.931} C_VEL
LIN {X 0,Y 410.053,Z 700.691,A -85,B 0,C 180,E1 -10535.409,E2 -10535.409} C_VEL
LIN {X 0,Y 410.19,Z 696.641,A -85,B 0,C 180,E1 -10536.888,E2 -10536.888} C_VEL
LIN {X 0,Y 410.476,Z 690.392,A -85,B 0,C 180,E1 -10538.616,E2 -10538.616} C_VEL
LIN {X 0,Y 410.876,Z 683.574,A -85,B 0,C 180,E1 -10540.098,E2 -10540.098} C_VEL
LIN {X 0,Y 411.325,Z 676.592,A -85,B 0,C 180,E1 -10541.332,E2 -10541.332} C_VEL
LIN {X 0,Y 411.95,Z 668.155,A -85,B 0,C 180,E1 -10542.563,E2 -10542.563} C_VEL
LIN {X 0,Y 412.676,Z 657.704,A -85,B 0,C 180,E1 -10543.794,E2 -10543.794} C_VEL
LIN {X 0,Y 413.321,Z 647.34,A -85,B 0,C 180,E1 -10544.777,E2 -10544.777} C_VEL
LIN {X 0,Y 414.065,Z 635.909,A -85,B 0,C 180,E1 -10545.632,E2 -10545.632} C_VEL
LIN {X 0,Y 414.742,Z 624.027,A -85,B 0,C 180,E1 -10546.3,E2 -10546.3} C_VEL
LIN {X 0,Y 415.263,Z 611.177,A -85,B 0,C 180,E1 -10546.816,E2 -10546.816} C_VEL
LIN {X 0,Y 416.081,Z 582.204,A -85,B 0,C 180,E1 -10547.542,E2 -10547.542} C_VEL
LIN {X 0,Y 417.524,Z 518.947,A -85,B 0,C 180,E1 -10548.981,E2 -10548.981} C_VEL
LIN {X 0,Y 415.375,Z 497.156,A -85,B 0,C 180,E1 -10549.677,E2 -10549.677} C_VEL
LIN {X 0,Y 412.891,Z 481.972,A -85,B 0,C 180,E1 -10550.259,E2 -10550.259} C_VEL
LIN {X 0,Y 414.319,Z 462.695,A -85,B 0,C 180,E1 -10553.653,E2 -10553.653} C_VEL
LIN {X 0,Y 415.884,Z 445.038,A -85,B 0,C 180,E1 -10556.887,E2 -10556.887} C_VEL
LIN {X 0,Y 415.845,Z 442.32,A -85,B 0,C 180,E1 -10557.422,E2 -10557.422} C_VEL
LIN {X 0,Y 413.997,Z 432.936,A -85,B 0,C 180,E1 -10559.492,E2 -10559.492} C_VEL
LIN {X 0,Y 411.217,Z 422.266,A -85,B 0,C 180,E1 -10562.155,E2 -10562.155} C_VEL
LIN {X 0,Y 411.199,Z 422.267,A -85,B 0,C 180,E1 -10565.529,E2 -10565.529} C_VEL
LIN {X 0,Y 411.212,Z 422.266,A -85,B 0,C 180,E1 -10569.225,E2 -10569.225} C_VEL
LIN {X 0,Y 411.179,Z 422.266,A -85,B 0,C 180,E1 -10572.695,E2 -10572.695} C_VEL
LIN {X 0,Y 411.17,Z 422.268,A -85,B 0,C 180,E1 -10575.881,E2 -10575.881} C_VEL
LIN {X 0,Y 411.166,Z 422.269,A -85,B 0,C 180,E1 -10578.772,E2 -10578.772} C_VEL
LIN {X 0,Y 411.208,Z 422.263,A -85,B 0,C 180,E1 -10581.831,E2 -10581.831} C_VEL
LIN {X 0,Y 411.213,Z 422.264,A -85,B 0,C 180,E1 -10585.122,E2 -10585.122} C_VEL
LIN {X 0,Y 411.168,Z 422.268,A -85,B 0,C 180,E1 -10588.003,E2 -10588.003} C_VEL
LIN {X 0,Y 411.22,Z 422.263,A -85,B 0,C 180,E1 -10591.41,E2 -10591.41} C_VEL
LIN {X 0,Y 411.239,Z 422.261,A -85,B 0,C 180,E1 -10593.619,E2 -10593.619} C_VEL
LIN {X 0,Y 411.205,Z 422.268,A -85,B 0,C 180,E1 -10596.853,E2 -10596.853} C_VEL
LIN {X 0,Y 411.237,Z 422.388,A -85,B 0,C 180,E1 -10599.762,E2 -10599.762} C_VEL
LIN {X 0,Y 412.251,Z 425.158,A -85,B 0,C 180,E1 -10599.923,E2 -10599.923} C_VEL
LIN {X 0,Y 417.669,Z 436.444,A -85,B 0,C 180,E1 -10600.636,E2 -10600.636} C_VEL
LIN {X 0,Y 418.998,Z 439.761,A -85,B 0,C 180,E1 -10600.821,E2 -10600.821} C_VEL
LIN {X 0,Y 417.159,Z 502.972,A -85,B 0,C 180,E1 -10602.32,E2 -10602.32} C_VEL
LIN {X 0,Y 416.659,Z 525.707,A -85,B 0,C 180,E1 -10602.863,E2 -10602.863} C_VEL
LIN {X 0,Y 416.331,Z 538.513,A -85,B 0,C 180,E1 -10603.355,E2 -10603.355} C_VEL
LIN {X 0,Y 415.946,Z 549.46,A -85,B 0,C 180,E1 -10603.938,E2 -10603.938} C_VEL
LIN {X 0,Y 415.333,Z 561.386,A -85,B 0,C 180,E1 -10604.767,E2 -10604.767} C_VEL
LIN {X 0,Y 414.596,Z 572.698,A -85,B 0,C 180,E1 -10605.771,E2 -10605.771} C_VEL
LIN {X 0,Y 414.038,Z 581.664,A -85,B 0,C 180,E1 -10606.753,E2 -10606.753} C_VEL
LIN {X 0,Y 413.286,Z 590.9,A -85,B 0,C 180,E1 -10607.976,E2 -10607.976} C_VEL
LIN {X 0,Y 412.629,Z 599.759,A -85,B 0,C 180,E1 -10609.45,E2 -10609.45} C_VEL
LIN {X 0,Y 412.088,Z 605.777,A -85,B 0,C 180,E1 -10610.676,E2 -10610.676} C_VEL
LIN {X 0,Y 411.573,Z 611.633,A -85,B 0,C 180,E1 -10612.148,E2 -10612.148} C_VEL
LIN {X 0,Y 411.096,Z 616.218,A -85,B 0,C 180,E1 -10613.62,E2 -10613.62} C_VEL
LIN {X 0,Y 411.006,Z 619.624,A -85,B 0,C 180,E1 -10615.095,E2 -10615.095} C_VEL
LIN {X 0,Y 410.768,Z 621.348,A -85,B 0,C 180,E1 -10616.076,E2 -10616.076} C_VEL
LIN {X 0,Y 410.506,Z 622.616,A -85,B 0,C 180,E1 -10617.056,E2 -10617.056} C_VEL
LIN {X 0,Y 410.335,Z 623.467,A -85,B 0,C 180,E1 -10618.037,E2 -10618.037} C_VEL
LIN {X 0,Y 410.261,Z 623.893,A -85,B 0,C 180,E1 -10619.018,E2 -10619.018} C_VEL
LIN {X 0,Y 410.225,Z 623.859,A -85,B 0,C 180,E1 -10620,E2 -10620} C_VEL
LIN {X 0,Y 410.231,Z 623.414,A -85,B 0,C 180,E1 -10620.982,E2 -10620.982} C_VEL
LIN {X 0,Y 410.312,Z 622.563,A -85,B 0,C 180,E1 -10621.963,E2 -10621.963} C_VEL
LIN {X 0,Y 410.492,Z 621.255,A -85,B 0,C 180,E1 -10622.944,E2 -10622.944} C_VEL
LIN {X 0,Y 410.679,Z 618.491,A -85,B 0,C 180,E1 -10624.417,E2 -10624.417} C_VEL
LIN {X 0,Y 410.717,Z 614.684,A -85,B 0,C 180,E1 -10625.893,E2 -10625.893} C_VEL
LIN {X 0,Y 411.046,Z 609.583,A -85,B 0,C 180,E1 -10627.397,E2 -10627.397} C_VEL
LIN {X 0,Y 411.316,Z 603.4,A -85,B 0,C 180,E1 -10628.846,E2 -10628.846} C_VEL
LIN {X 0,Y 411.818,Z 595.558,A -85,B 0,C 180,E1 -10630.323,E2 -10630.323} C_VEL
LIN {X 0,Y 412.259,Z 587.532,A -85,B 0,C 180,E1 -10631.555,E2 -10631.555} C_VEL
LIN {X 0,Y 412.89,Z 576.621,A -85,B 0,C 180,E1 -10632.909,E2 -10632.909} C_VEL
LIN {X 0,Y 413.414,Z 566.7,A -85,B 0,C 180,E1 -10633.907,E2 -10633.907} C_VEL
LIN {X 0,Y 413.913,Z 554.593,A -85,B 0,C 180,E1 -10634.881,E2 -10634.881} C_VEL
LIN {X 0,Y 414.357,Z 541.62,A -85,B 0,C 180,E1 -10635.683,E2 -10635.683} C_VEL
LIN {X 0,Y 414.766,Z 528.511,A -85,B 0,C 180,E1 -10636.267,E2 -10636.267} C_VEL
LIN {X 0,Y 414.986,Z 514.753,A -85,B 0,C 180,E1 -10636.669,E2 -10636.669} C_VEL
LIN {X 0,Y 416.388,Z 438.029,A -85,B 0,C 180,E1 -10638.259,E2 -10638.259} C_VEL
LIN {X 0,Y 411.268,Z 422.259,A -85,B 0,C 180,E1 -10638.822,E2 -10638.822} C_VEL
LIN {X 0,Y 411.204,Z 422.26,A -85,B 0,C 180,E1 -10642.641,E2 -10642.641} C_VEL
LIN {X 0,Y 411.236,Z 422.262,A -85,B 0,C 180,E1 -10645.293,E2 -10645.293} C_VEL
LIN {X 0,Y 411.261,Z 422.253,A -85,B 0,C 180,E1 -10647.478,E2 -10647.478} C_VEL
LIN {X 0,Y 411.192,Z 422.266,A -85,B 0,C 180,E1 -10650.848,E2 -10650.848} C_VEL
LIN {X 0,Y 411.208,Z 422.246,A -85,B 0,C 180,E1 -10654.334,E2 -10654.334} C_VEL
LIN {X 0,Y 411.196,Z 422.264,A -85,B 0,C 180,E1 -10657.974,E2 -10657.974} C_VEL
LIN {X 0,Y 411.166,Z 422.262,A -85,B 0,C 180,E1 -10661.228,E2 -10661.228} C_VEL
LIN {X 0,Y 411.178,Z 422.269,A -85,B 0,C 180,E1 -10664.49,E2 -10664.49} C_VEL
LIN {X 0,Y 411.18,Z 422.266,A -85,B 0,C 180,E1 -10668.195,E2 -10668.195} C_VEL
LIN {X 0,Y 411.216,Z 422.26,A -85,B 0,C 180,E1 -10670.775,E2 -10670.775} C_VEL
LIN {X 0,Y 411.2,Z 422.266,A -85,B 0,C 180,E1 -10674.471,E2 -10674.471} C_VEL
LIN {X 0,Y 411.21,Z 422.265,A -85,B 0,C 180,E1 -10676.873,E2 -10676.873} C_VEL
LIN {X 0,Y 411.213,Z 422.271,A -85,B 0,C 180,E1 -10680.65,E2 -10680.65} C_VEL
LIN {X 0,Y 411.21,Z 422.304,A -85,B 0,C 180,E1 -10681.931,E2 -10681.931} C_VEL
LIN {X 0,Y 414.516,Z 437.722,A -85,B 0,C 180,E1 -10684.921,E2 -10684.921} C_VEL
LIN {X 0,Y 414.821,Z 442.218,A -85,B 0,C 180,E1 -10685.742,E2 -10685.742} C_VEL
LIN {X 0,Y 414.038,Z 460.422,A -85,B 0,C 180,E1 -10688.883,E2 -10688.883} C_VEL
LIN {X 0,Y 413.638,Z 471.666,A -85,B 0,C 180,E1 -10690.703,E2 -10690.703} C_VEL
LIN {X 0,Y 417.2,Z 492.638,A -85,B 0,C 180,E1 -10691.253,E2 -10691.253} C_VEL
LIN {X 0,Y 416.215,Z 577.024,A -85,B 0,C 180,E1 -10692.718,E2 -10692.718} C_VEL
LIN {X 0,Y 415.917,Z 589.831,A -85,B 0,C 180,E1 -10693.053,E2 -10693.053} C_VEL
LIN {X 0,Y 415.714,Z 596.234,A -85,B 0,C 180,E1 -10693.297,E2 -10693.297} C_VEL
LIN {X 0,Y 414.859,Z 600.012,A -85,B 0,C 180,E1 -10693.432,E2 -10693.432} C_VEL
LIN {X 0,Y 408.717,Z 611.708,A -85,B 0,C 180,E1 -10693.837,E2 -10693.837} C_VEL
LIN {X 0,Y 407.909,Z 615.296,A -85,B 0,C 180,E1 -10694.051,E2 -10694.051} C_VEL
LIN {X 0,Y 407.255,Z 625.856,A -85,B 0,C 180,E1 -10694.87,E2 -10694.87} C_VEL
LIN {X 0,Y 406.555,Z 637.198,A -85,B 0,C 180,E1 -10695.995,E2 -10695.995} C_VEL
LIN {X 0,Y 405.641,Z 647.329,A -85,B 0,C 180,E1 -10697.238,E2 -10697.238} C_VEL
LIN {X 0,Y 404.906,Z 655.547,A -85,B 0,C 180,E1 -10698.486,E2 -10698.486} C_VEL
LIN {X 0,Y 404.308,Z 663.559,A -85,B 0,C 180,E1 -10699.989,E2 -10699.989} C_VEL
LIN {X 0,Y 403.715,Z 670.009,A -85,B 0,C 180,E1 -10701.491,E2 -10701.491} C_VEL
LIN {X 0,Y 403.366,Z 675.971,A -85,B 0,C 180,E1 -10703.283,E2 -10703.283} C_VEL
LIN {X 0,Y 403.104,Z 680.177,A -85,B 0,C 180,E1 -10704.999,E2 -10704.999} C_VEL
LIN {X 0,Y 402.957,Z 682.038,A -85,B 0,C 180,E1 -10706,E2 -10706} C_VEL
LIN {X 0,Y 402.942,Z 683.459,A -85,B 0,C 180,E1 -10707.001,E2 -10707.001} C_VEL
LIN {X 0,Y 402.925,Z 684.454,A -85,B 0,C 180,E1 -10708.001,E2 -10708.001} C_VEL
LIN {X 0,Y 402.851,Z 685.306,A -85,B 0,C 180,E1 -10710,E2 -10710} C_VEL
LIN {X 0,Y 402.867,Z 685.115,A -85,B 0,C 180,E1 -10711,E2 -10711} C_VEL
LIN {X 0,Y 402.925,Z 684.528,A -85,B 0,C 180,E1 -10711.999,E2 -10711.999} C_VEL
LIN {X 0,Y 402.942,Z 683.563,A -85,B 0,C 180,E1 -10712.999,E2 -10712.999} C_VEL
LIN {X 0,Y 402.956,Z 682.2,A -85,B 0,C 180,E1 -10714,E2 -10714} C_VEL
LIN {X 0,Y 403.188,Z 679.329,A -85,B 0,C 180,E1 -10715.501,E2 -10715.501} C_VEL
LIN {X 0,Y 403.365,Z 675.432,A -85,B 0,C 180,E1 -10717.006,E2 -10717.006} C_VEL
LIN {X 0,Y 403.713,Z 670.38,A -85,B 0,C 180,E1 -10718.509,E2 -10718.509} C_VEL
LIN {X 0,Y 404.244,Z 664.009,A -85,B 0,C 180,E1 -10720.012,E2 -10720.012} C_VEL
LIN {X 0,Y 404.895,Z 656.094,A -85,B 0,C 180,E1 -10721.514,E2 -10721.514} C_VEL
LIN {X 0,Y 405.614,Z 648.005,A -85,B 0,C 180,E1 -10722.763,E2 -10722.763} C_VEL
LIN {X 0,Y 406.44,Z 638.064,A -85,B 0,C 180,E1 -10724.01,E2 -10724.01} C_VEL
LIN {X 0,Y 407.179,Z 626.892,A -85,B 0,C 180,E1 -10725.133,E2 -10725.133} C_VEL
LIN {X 0,Y 407.881,Z 615.95,A -85,B 0,C 180,E1 -10726.003,E2 -10726.003} C_VEL
LIN {X 0,Y 408.558,Z 604.851,A -85,B 0,C 180,E1 -10726.682,E2 -10726.682} C_VEL
LIN {X 0,Y 409.11,Z 591.66,A -85,B 0,C 180,E1 -10727.27,E2 -10727.27} C_VEL
LIN {X 0,Y 409.461,Z 580.042,A -85,B 0,C 180,E1 -10727.609,E2 -10727.609} C_VEL
LIN {X 0,Y 410.537,Z 493.366,A -85,B 0,C 180,E1 -10729.149,E2 -10729.149} C_VEL
LIN {X 0,Y 406.839,Z 471.608,A -85,B 0,C 180,E1 -10729.756,E2 -10729.756} C_VEL
LIN {X 0,Y 407.47,Z 454.796,A -85,B 0,C 180,E1 -10732.567,E2 -10732.567} C_VEL
LIN {X 0,Y 408.066,Z 442.718,A -85,B 0,C 180,E1 -10734.686,E2 -10734.686} C_VEL
LIN {X 0,Y 406.678,Z 434.508,A -85,B 0,C 180,E1 -10736.26,E2 -10736.26} C_VEL
LIN {X 0,Y 404.16,Z 423.142,A -85,B 0,C 180,E1 -10738.497,E2 -10738.497} C_VEL
LIN {X 0,Y 404.142,Z 423.147,A -85,B 0,C 180,E1 -10741.558,E2 -10741.558} C_VEL
LIN {X 0,Y 404.187,Z 423.139,A -85,B 0,C 180,E1 -10745.016,E2 -10745.016} C_VEL
LIN {X 0,Y 404.155,Z 423.142,A -85,B 0,C 180,E1 -10748.757,E2 -10748.757} C_VEL
LIN {X 0,Y 404.126,Z 423.147,A -85,B 0,C 180,E1 -10751.6,E2 -10751.6} C_VEL
LIN {X 0,Y 404.149,Z 423.138,A -85,B 0,C 180,E1 -10754.522,E2 -10754.522} C_VEL
LIN {X 0,Y 404.142,Z 423.139,A -85,B 0,C 180,E1 -10757.296,E2 -10757.296} C_VEL
LIN {X 0,Y 404.171,Z 423.138,A -85,B 0,C 180,E1 -10759.955,E2 -10759.955} C_VEL
LIN {X 0,Y 404.138,Z 423.131,A -85,B 0,C 180,E1 -10763.125,E2 -10763.125} C_VEL
LIN {X 0,Y 404.147,Z 423.141,A -85,B 0,C 180,E1 -10766.188,E2 -10766.188} C_VEL
LIN {X 0,Y 404.146,Z 423.142,A -85,B 0,C 180,E1 -10769.715,E2 -10769.715} C_VEL
LIN {X 0,Y 404.217,Z 423.216,A -85,B 0,C 180,E1 -10772.067,E2 -10772.067} C_VEL
LIN {X 0,Y 407.344,Z 438.759,A -85,B 0,C 180,E1 -10774.994,E2 -10774.994} C_VEL
LIN {X 0,Y 407.672,Z 443.709,A -85,B 0,C 180,E1 -10775.878,E2 -10775.878} C_VEL
LIN {X 0,Y 406.765,Z 463.632,A -85,B 0,C 180,E1 -10779.334,E2 -10779.334} C_VEL
LIN {X 0,Y 406.368,Z 472.212,A -85,B 0,C 180,E1 -10780.816,E2 -10780.816} C_VEL
LIN {X 0,Y 409.438,Z 492.746,A -85,B 0,C 180,E1 -10781.4,E2 -10781.4} C_VEL
LIN {X 0,Y 407.78,Z 583.374,A -85,B 0,C 180,E1 -10783.35,E2 -10783.35} C_VEL
LIN {X 0,Y 407.345,Z 596.798,A -85,B 0,C 180,E1 -10783.847,E2 -10783.847} C_VEL
LIN {X 0,Y 406.861,Z 608.683,A -85,B 0,C 180,E1 -10784.47,E2 -10784.47} C_VEL
LIN {X 0,Y 406.184,Z 621.683,A -85,B 0,C 180,E1 -10785.38,E2 -10785.38} C_VEL
LIN {X 0,Y 405.693,Z 632.465,A -85,B 0,C 180,E1 -10786.347,E2 -10786.347} C_VEL
LIN {X 0,Y 404.992,Z 643.649,A -85,B 0,C 180,E1 -10787.599,E2 -10787.599} C_VEL
LIN {X 0,Y 404.478,Z 651.889,A -85,B 0,C 180,E1 -10788.727,E2 -10788.727} C_VEL
LIN {X 0,Y 403.914,Z 660.824,A -85,B 0,C 180,E1 -10790.233,E2 -10790.233} C_VEL
LIN {X 0,Y 403.48,Z 668.024,A -85,B 0,C 180,E1 -10791.738,E2 -10791.738} C_VEL
LIN {X 0,Y 403.277,Z 672.87,A -85,B 0,C 180,E1 -10792.993,E2 -10792.993} C_VEL
LIN {X 0,Y 403.116,Z 677.533,A -85,B 0,C 180,E1 -10794.497,E2 -10794.497} C_VEL
LIN {X 0,Y 402.932,Z 681.025,A -85,B 0,C 180,E1 -10795.999,E2 -10795.999} C_VEL
LIN {X 0,Y 402.901,Z 682.742,A -85,B 0,C 180,E1 -10797,E2 -10797} C_VEL
LIN {X 0,Y 402.921,Z 684.043,A -85,B 0,C 180,E1 -10798.001,E2 -10798.001} C_VEL
LIN {X 0,Y 402.867,Z 684.904,A -85,B 0,C 180,E1 -10799,E2 -10799} C_VEL
LIN {X 0,Y 402.851,Z 685.311,A -85,B 0,C 180,E1 -10800,E2 -10800} C_VEL
LIN {X 0,Y 402.867,Z 685.313,A -85,B 0,C 180,E1 -10801,E2 -10801} C_VEL
LIN {X 0,Y 402.946,Z 684.875,A -85,B 0,C 180,E1 -10801.999,E2 -10801.999} C_VEL
LIN {X 0,Y 402.99,Z 683.985,A -85,B 0,C 180,E1 -10802.999,E2 -10802.999} C_VEL
LIN {X 0,Y 402.963,Z 682.69,A -85,B 0,C 180,E1 -10804,E2 -10804} C_VEL
LIN {X 0,Y 403.229,Z 679.884,A -85,B 0,C 180,E1 -10805.501,E2 -10805.501} C_VEL
LIN {X 0,Y 403.391,Z 676.009,A -85,B 0,C 180,E1 -10807.005,E2 -10807.005} C_VEL
LIN {X 0,Y 403.777,Z 670.919,A -85,B 0,C 180,E1 -10808.508,E2 -10808.508} C_VEL
LIN {X 0,Y 404.279,Z 664.48,A -85,B 0,C 180,E1 -10810.011,E2 -10810.011} C_VEL
LIN {X 0,Y 404.974,Z 656.451,A -85,B 0,C 180,E1 -10811.512,E2 -10811.512} C_VEL
LIN {X 0,Y 405.599,Z 648.184,A -85,B 0,C 180,E1 -10812.763,E2 -10812.763} C_VEL
LIN {X 0,Y 406.403,Z 638.126,A -85,B 0,C 180,E1 -10814.011,E2 -10814.011} C_VEL
LIN {X 0,Y 407.225,Z 626.92,A -85,B 0,C 180,E1 -10815.131,E2 -10815.131} C_VEL
LIN {X 0,Y 408.04,Z 614.267,A -85,B 0,C 180,E1 -10816.125,E2 -10816.125} C_VEL
LIN {X 0,Y 408.768,Z 601.705,A -85,B 0,C 180,E1 -10816.866,E2 -10816.866} C_VEL
LIN {X 0,Y 409.357,Z 587.966,A -85,B 0,C 180,E1 -10817.452,E2 -10817.452} C_VEL
LIN {X 0,Y 409.87,Z 572.92,A -85,B 0,C 180,E1 -10817.848,E2 -10817.848} C_VEL
LIN {X 0,Y 412.071,Z 498.322,A -85,B 0,C 180,E1 -10819.621,E2 -10819.621} C_VEL
LIN {X 0,Y 412.036,Z 492.32,A -85,B 0,C 180,E1 -10819.786,E2 -10819.786} C_VEL
LIN {X 0,Y 409.316,Z 478.159,A -85,B 0,C 180,E1 -10820.375,E2 -10820.375} C_VEL
LIN {X 0,Y 408.348,Z 473.789,A -85,B 0,C 180,E1 -10820.601,E2 -10820.601} C_VEL
LIN {X 0,Y 409.54,Z 453.896,A -85,B 0,C 180,E1 -10824.052,E2 -10824.052} C_VEL
LIN {X 0,Y 409.887,Z 446.29,A -85,B 0,C 180,E1 -10825.382,E2 -10825.382} C_VEL
LIN {X 0,Y 408.332,Z 437.503,A -85,B 0,C 180,E1 -10827.135,E2 -10827.135} C_VEL
LIN {X 0,Y 405.956,Z 428.731,A -85,B 0,C 180,E1 -10828.996,E2 -10828.996} C_VEL
LIN {X 0,Y 404.146,Z 423.148,A -85,B 0,C 180,E1 -10830.285,E2 -10830.285} C_VEL
LIN {X 0,Y 404.147,Z 423.144,A -85,B 0,C 180,E1 -10833.812,E2 -10833.812} C_VEL
LIN {X 0,Y 404.138,Z 423.143,A -85,B 0,C 180,E1 -10836.875,E2 -10836.875} C_VEL
LIN {X 0,Y 404.149,Z 423.142,A -85,B 0,C 180,E1 -10840.08,E2 -10840.08} C_VEL
LIN {X 0,Y 404.155,Z 423.141,A -85,B 0,C 180,E1 -10843.084,E2 -10843.084} C_VEL
LIN {X 0,Y 404.15,Z 423.143,A -85,B 0,C 180,E1 -10845.926,E2 -10845.926} C_VEL
LIN {X 0,Y 404.121,Z 423.145,A -85,B 0,C 180,E1 -10848.635,E2 -10848.635} C_VEL
LIN {X 0,Y 404.155,Z 423.141,A -85,B 0,C 180,E1 -10851.492,E2 -10851.492} C_VEL
LIN {X 0,Y 404.186,Z 423.138,A -85,B 0,C 180,E1 -10854.984,E2 -10854.984} C_VEL
LIN {X 0,Y 404.144,Z 423.145,A -85,B 0,C 180,E1 -10858.554,E2 -10858.554} C_VEL
LIN {X 0,Y 404.21,Z 423.285,A -85,B 0,C 180,E1 -10859.214,E2 -10859.214} C_VEL
LIN {X 0,Y 407.933,Z 440.866,A -85,B 0,C 180,E1 -10862.557,E2 -10862.557} C_VEL
LIN {X 0,Y 408.206,Z 445.624,A -85,B 0,C 180,E1 -10863.408,E2 -10863.408} C_VEL
LIN {X 0,Y 406.733,Z 467.279,A -85,B 0,C 180,E1 -10867.121,E2 -10867.121} C_VEL
LIN {X 0,Y 405.981,Z 480.611,A -85,B 0,C 180,E1 -10869.349,E2 -10869.349} C_VEL
LIN {X 0,Y 406.85,Z 487.257,A -85,B 0,C 180,E1 -10869.699,E2 -10869.699} C_VEL
LIN {X 0,Y 408.814,Z 501.778,A -85,B 0,C 180,E1 -10870.267,E2 -10870.267} C_VEL
LIN {X 0,Y 410.557,Z 521.143,A -85,B 0,C 180,E1 -10870.922,E2 -10870.922} C_VEL
LIN {X 0,Y 409.279,Z 565.315,A -85,B 0,C 180,E1 -10871.996,E2 -10871.996} C_VEL
LIN {X 0,Y 408.655,Z 604.923,A -85,B 0,C 180,E1 -10872.71,E2 -10872.71} C_VEL
LIN {X 0,Y 408.149,Z 618.606,A -85,B 0,C 180,E1 -10873.172,E2 -10873.172} C_VEL
LIN {X 0,Y 407.539,Z 630.906,A -85,B 0,C 180,E1 -10873.79,E2 -10873.79} C_VEL
LIN {X 0,Y 406.777,Z 642.672,A -85,B 0,C 180,E1 -10874.595,E2 -10874.595} C_VEL
LIN {X 0,Y 405.981,Z 654.472,A -85,B 0,C 180,E1 -10875.641,E2 -10875.641} C_VEL
LIN {X 0,Y 405.228,Z 664.32,A -85,B 0,C 180,E1 -10876.739,E2 -10876.739} C_VEL
LIN {X 0,Y 404.589,Z 673.252,A -85,B 0,C 180,E1 -10877.968,E2 -10877.968} C_VEL
LIN {X 0,Y 403.907,Z 682.111,A -85,B 0,C 180,E1 -10879.473,E2 -10879.473} C_VEL
LIN {X 0,Y 403.482,Z 689.212,A -85,B 0,C 180,E1 -10880.981,E2 -10880.981} C_VEL
LIN {X 0,Y 403.148,Z 694.852,A -85,B 0,C 180,E1 -10882.487,E2 -10882.487} C_VEL
LIN {X 0,Y 402.987,Z 699.268,A -85,B 0,C 180,E1 -10883.994,E2 -10883.994} C_VEL
LIN {X 0,Y 402.924,Z 703.569,A -85,B 0,C 180,E1 -10885.999,E2 -10885.999} C_VEL
LIN {X 0,Y 402.91,Z 705.018,A -85,B 0,C 180,E1 -10887,E2 -10887} C_VEL
LIN {X 0,Y 402.937,Z 706.032,A -85,B 0,C 180,E1 -10888.001,E2 -10888.001} C_VEL
LIN {X 0,Y 402.907,Z 706.768,A -85,B 0,C 180,E1 -10890,E2 -10890} C_VEL
LIN {X 0,Y 402.91,Z 706.546,A -85,B 0,C 180,E1 -10890.999,E2 -10890.999} C_VEL
LIN {X 0,Y 402.939,Z 705.929,A -85,B 0,C 180,E1 -10891.999,E2 -10891.999} C_VEL
LIN {X 0,Y 402.916,Z 704.919,A -85,B 0,C 180,E1 -10893,E2 -10893} C_VEL
LIN {X 0,Y 402.932,Z 703.485,A -85,B 0,C 180,E1 -10894.001,E2 -10894.001} C_VEL
LIN {X 0,Y 402.953,Z 700.501,A -85,B 0,C 180,E1 -10895.505,E2 -10895.505} C_VEL
LIN {X 0,Y 403.108,Z 696.451,A -85,B 0,C 180,E1 -10897.01,E2 -10897.01} C_VEL
LIN {X 0,Y 403.415,Z 690.203,A -85,B 0,C 180,E1 -10898.768,E2 -10898.768} C_VEL
LIN {X 0,Y 403.853,Z 683.386,A -85,B 0,C 180,E1 -10900.275,E2 -10900.275} C_VEL
LIN {X 0,Y 404.338,Z 676.406,A -85,B 0,C 180,E1 -10901.53,E2 -10901.53} C_VEL
LIN {X 0,Y 404.992,Z 667.97,A -85,B 0,C 180,E1 -10902.783,E2 -10902.783} C_VEL
LIN {X 0,Y 405.768,Z 657.049,A -85,B 0,C 180,E1 -10904.085,E2 -10904.085} C_VEL
LIN {X 0,Y 406.564,Z 645.729,A -85,B 0,C 180,E1 -10905.157,E2 -10905.157} C_VEL
LIN {X 0,Y 407.343,Z 633.771,A -85,B 0,C 180,E1 -10906.025,E2 -10906.025} C_VEL
LIN {X 0,Y 408.026,Z 621.296,A -85,B 0,C 180,E1 -10906.704,E2 -10906.704} C_VEL
LIN {X 0,Y 408.566,Z 609.14,A -85,B 0,C 180,E1 -10907.165,E2 -10907.165} C_VEL
LIN {X 0,Y 409.383,Z 584.846,A -85,B 0,C 180,E1 -10907.838,E2 -10907.838} C_VEL
LIN {X 0,Y 411.129,Z 520.581,A -85,B 0,C 180,E1 -10909.338,E2 -10909.338} C_VEL
LIN {X 0,Y 409.061,Z 498.873,A -85,B 0,C 180,E1 -10910.058,E2 -10910.058} C_VEL
LIN {X 0,Y 406.157,Z 480.875,A -85,B 0,C 180,E1 -10910.789,E2 -10910.789} C_VEL
LIN {X 0,Y 407.577,Z 462.612,A -85,B 0,C 180,E1 -10914.093,E2 -10914.093} C_VEL
LIN {X 0,Y 409.126,Z 446.753,A -85,B 0,C 180,E1 -10917.079,E2 -10917.079} C_VEL
LIN {X 0,Y 409.08,Z 444.01,A -85,B 0,C 180,E1 -10917.637,E2 -10917.637} C_VEL
LIN {X 0,Y 407.243,Z 434.804,A -85,B 0,C 180,E1 -10919.746,E2 -10919.746} C_VEL
LIN {X 0,Y 404.861,Z 425.771,A -85,B 0,C 180,E1 -10922.054,E2 -10922.054} C_VEL
LIN {X 0,Y 404.179,Z 423.141,A -85,B 0,C 180,E1 -10922.818,E2 -10922.818} C_VEL
LIN {X 0,Y 404.143,Z 423.144,A -85,B 0,C 180,E1 -10926.246,E2 -10926.246} C_VEL
LIN {X 0,Y 404.152,Z 423.142,A -85,B 0,C 180,E1 -10928.757,E2 -10928.757} C_VEL
LIN {X 0,Y 404.121,Z 423.148,A -85,B 0,C 180,E1 -10931.599,E2 -10931.599} C_VEL
LIN {X 0,Y 404.147,Z 423.143,A -85,B 0,C 180,E1 -10934.522,E2 -10934.522} C_VEL
LIN {X 0,Y 404.139,Z 423.147,A -85,B 0,C 180,E1 -10937.296,E2 -10937.296} C_VEL
LIN {X 0,Y 404.171,Z 423.139,A -85,B 0,C 180,E1 -10939.955,E2 -10939.955} C_VEL
LIN {X 0,Y 404.139,Z 423.143,A -85,B 0,C 180,E1 -10943.125,E2 -10943.125} C_VEL
LIN {X 0,Y 404.147,Z 423.141,A -85,B 0,C 180,E1 -10946.188,E2 -10946.188} C_VEL
LIN {X 0,Y 404.148,Z 423.143,A -85,B 0,C 180,E1 -10949.715,E2 -10949.715} C_VEL
LIN {X 0,Y 404.197,Z 423.141,A -85,B 0,C 180,E1 -10953.123,E2 -10953.123} C_VEL
LIN {X 0,Y 404.179,Z 423.144,A -85,B 0,C 180,E1 -10955.334,E2 -10955.334} C_VEL
LIN {X 0,Y 404.141,Z 423.147,A -85,B 0,C 180,E1 -10958.581,E2 -10958.581} C_VEL
LIN {X 0,Y 404.178,Z 423.142,A -85,B 0,C 180,E1 -10959.193,E2 -10959.193} C_VEL
LIN {X 0,Y 405.26,Z 426.125,A -85,B 0,C 180,E1 -10959.379,E2 -10959.379} C_VEL
LIN {X 0,Y 410.751,Z 437.204,A -85,B 0,C 180,E1 -10960.149,E2 -10960.149} C_VEL
LIN {X 0,Y 412.677,Z 442.169,A -85,B 0,C 180,E1 -10960.434,E2 -10960.434} C_VEL
LIN {X 0,Y 410.134,Z 525.904,A -85,B 0,C 180,E1 -10962.485,E2 -10962.485} C_VEL
LIN {X 0,Y 409.741,Z 538.83,A -85,B 0,C 180,E1 -10962.983,E2 -10962.983} C_VEL
LIN {X 0,Y 409.288,Z 551.411,A -85,B 0,C 180,E1 -10963.669,E2 -10963.669} C_VEL
LIN {X 0,Y 408.595,Z 563.569,A -85,B 0,C 180,E1 -10964.552,E2 -10964.552} C_VEL
LIN {X 0,Y 407.862,Z 574.235,A -85,B 0,C 180,E1 -10965.531,E2 -10965.531} C_VEL
LIN {X 0,Y 407.25,Z 583.04,A -85,B 0,C 180,E1 -10966.528,E2 -10966.528} C_VEL
LIN {X 0,Y 406.464,Z 592.096,A -85,B 0,C 180,E1 -10967.772,E2 -10967.772} C_VEL
LIN {X 0,Y 405.734,Z 600.86,A -85,B 0,C 180,E1 -10969.268,E2 -10969.268} C_VEL
LIN {X 0,Y 405.155,Z 606.831,A -85,B 0,C 180,E1 -10970.515,E2 -10970.515} C_VEL
LIN {X 0,Y 404.612,Z 612.641,A -85,B 0,C 180,E1 -10972.012,E2 -10972.012} C_VEL
LIN {X 0,Y 404.116,Z 617.176,A -85,B 0,C 180,E1 -10973.509,E2 -10973.509} C_VEL
LIN {X 0,Y 403.988,Z 620.532,A -85,B 0,C 180,E1 -10975.01,E2 -10975.01} C_VEL
LIN {X 0,Y 403.742,Z 622.197,A -85,B 0,C 180,E1 -10976.007,E2 -10976.007} C_VEL
LIN {X 0,Y 403.468,Z 623.431,A -85,B 0,C 180,E1 -10977.005,E2 -10977.005} C_VEL
LIN {X 0,Y 403.286,Z 624.25,A -85,B 0,C 180,E1 -10978.003,E2 -10978.003} C_VEL
LIN {X 0,Y 403.202,Z 624.625,A -85,B 0,C 180,E1 -10979.001,E2 -10979.001} C_VEL
LIN {X 0,Y 403.165,Z 624.553,A -85,B 0,C 180,E1 -10980,E2 -10980} C_VEL
LIN {X 0,Y 403.174,Z 624.077,A -85,B 0,C 180,E1 -10980.999,E2 -10980.999} C_VEL
LIN {X 0,Y 403.264,Z 623.189,A -85,B 0,C 180,E1 -10981.998,E2 -10981.998} C_VEL
LIN {X 0,Y 403.451,Z 621.828,A -85,B 0,C 180,E1 -10982.996,E2 -10982.996} C_VEL
LIN {X 0,Y 403.626,Z 618.997,A -85,B 0,C 180,E1 -10984.494,E2 -10984.494} C_VEL
LIN {X 0,Y 403.667,Z 615.112,A -85,B 0,C 180,E1 -10985.996,E2 -10985.996} C_VEL
LIN {X 0,Y 404.033,Z 609.237,A -85,B 0,C 180,E1 -10987.706,E2 -10987.706} C_VEL
LIN {X 0,Y 404.371,Z 602.447,A -85,B 0,C 180,E1 -10989.251,E2 -10989.251} C_VEL
LIN {X 0,Y 404.892,Z 594.133,A -85,B 0,C 180,E1 -10990.754,E2 -10990.754} C_VEL
LIN {X 0,Y 405.369,Z 585.649,A -85,B 0,C 180,E1 -10992.008,E2 -10992.008} C_VEL
LIN {X 0,Y 406.019,Z 575.275,A -85,B 0,C 180,E1 -10993.259,E2 -10993.259} C_VEL
LIN {X 0,Y 406.623,Z 563.492,A -85,B 0,C 180,E1 -10994.391,E2 -10994.391} C_VEL
LIN {X 0,Y 407.059,Z 552.07,A -85,B 0,C 180,E1 -10995.266,E2 -10995.266} C_VEL
LIN {X 0,Y 407.525,Z 539.12,A -85,B 0,C 180,E1 -10996.018,E2 -10996.018} C_VEL
LIN {X 0,Y 407.927,Z 525.632,A -85,B 0,C 180,E1 -10996.58,E2 -10996.58} C_VEL
LIN {X 0,Y 408.114,Z 510.977,A -85,B 0,C 180,E1 -10996.958,E2 -10996.958} C_VEL
LIN {X 0,Y 409.341,Z 438.527,A -85,B 0,C 180,E1 -10998.503,E2 -10998.503} C_VEL
LIN {X 0,Y 404.204,Z 423.171,A -85,B 0,C 180,E1 -10999.054,E2 -10999.054} C_VEL
LIN {X 0,Y 404.153,Z 423.139,A -85,B 0,C 180,E1 -11002.832,E2 -11002.832} C_VEL
LIN {X 0,Y 404.183,Z 423.137,A -85,B 0,C 180,E1 -11005.767,E2 -11005.767} C_VEL
LIN {X 0,Y 404.197,Z 423.131,A -85,B 0,C 180,E1 -11008,E2 -11008} C_VEL
LIN {X 0,Y 404.142,Z 423.136,A -85,B 0,C 180,E1 -11011.558,E2 -11011.558} C_VEL
LIN {X 0,Y 404.187,Z 423.126,A -85,B 0,C 180,E1 -11015.016,E2 -11015.016} C_VEL
LIN {X 0,Y 404.155,Z 423.141,A -85,B 0,C 180,E1 -11018.757,E2 -11018.757} C_VEL
LIN {X 0,Y 404.126,Z 423.143,A -85,B 0,C 180,E1 -11021.6,E2 -11021.6} C_VEL
LIN {X 0,Y 404.148,Z 423.143,A -85,B 0,C 180,E1 -11024.522,E2 -11024.522} C_VEL
LIN {X 0,Y 404.139,Z 423.143,A -85,B 0,C 180,E1 -11027.296,E2 -11027.296} C_VEL
LIN {X 0,Y 404.171,Z 423.132,A -85,B 0,C 180,E1 -11029.955,E2 -11029.955} C_VEL
LIN {X 0,Y 404.138,Z 423.139,A -85,B 0,C 180,E1 -11033.125,E2 -11033.125} C_VEL
LIN {X 0,Y 404.147,Z 423.14,A -85,B 0,C 180,E1 -11036.188,E2 -11036.188} C_VEL
LIN {X 0,Y 404.146,Z 423.146,A -85,B 0,C 180,E1 -11039.715,E2 -11039.715} C_VEL
LIN {X 0,Y 404.201,Z 423.329,A -85,B 0,C 180,E1 -11041.647,E2 -11041.647} C_VEL
LIN {X 0,Y 407.608,Z 439.051,A -85,B 0,C 180,E1 -11044.739,E2 -11044.739} C_VEL
LIN {X 0,Y 408.034,Z 442.053,A -85,B 0,C 180,E1 -11045.311,E2 -11045.311} C_VEL
LIN {X 0,Y 407.211,Z 460.291,A -85,B 0,C 180,E1 -11048.485,E2 -11048.485} C_VEL
LIN {X 0,Y 406.773,Z 471.756,A -85,B 0,C 180,E1 -11050.364,E2 -11050.364} C_VEL
LIN {X 0,Y 410.491,Z 493.66,A -85,B 0,C 180,E1 -11050.951,E2 -11050.951} C_VEL
LIN {X 0,Y 409.464,Z 577.129,A -85,B 0,C 180,E1 -11052.423,E2 -11052.423} C_VEL
LIN {X 0,Y 409.153,Z 589.98,A -85,B 0,C 180,E1 -11052.764,E2 -11052.764} C_VEL
LIN {X 0,Y 408.579,Z 603.015,A -85,B 0,C 180,E1 -11053.319,E2 -11053.319} C_VEL
LIN {X 0,Y 407.909,Z 615.296,A -85,B 0,C 180,E1 -11054.051,E2 -11054.051} C_VEL
LIN {X 0,Y 407.019,Z 620.56,A -85,B 0,C 180,E1 -11054.41,E2 -11054.41} C_VEL
LIN {X 0,Y 403.762,Z 628.885,A -85,B 0,C 180,E1 -11055.01,E2 -11055.01} C_VEL
LIN {X 0,Y 400.392,Z 636.825,A -85,B 0,C 180,E1 -11055.71,E2 -11055.71} C_VEL
LIN {X 0,Y 399.333,Z 641.398,A -85,B 0,C 180,E1 -11056.22,E2 -11056.22} C_VEL
LIN {X 0,Y 398.388,Z 650.989,A -85,B 0,C 180,E1 -11057.52,E2 -11057.52} C_VEL
LIN {X 0,Y 397.728,Z 658.622,A -85,B 0,C 180,E1 -11058.792,E2 -11058.792} C_VEL
LIN {X 0,Y 397.091,Z 666.061,A -85,B 0,C 180,E1 -11060.32,E2 -11060.32} C_VEL
LIN {X 0,Y 396.534,Z 672.032,A -85,B 0,C 180,E1 -11061.849,E2 -11061.849} C_VEL
LIN {X 0,Y 396.29,Z 676.486,A -85,B 0,C 180,E1 -11063.283,E2 -11063.283} C_VEL
LIN {X 0,Y 396.049,Z 680.365,A -85,B 0,C 180,E1 -11064.91,E2 -11064.91} C_VEL
LIN {X 0,Y 395.88,Z 682.227,A -85,B 0,C 180,E1 -11065.928,E2 -11065.928} C_VEL
LIN {X 0,Y 395.846,Z 683.648,A -85,B 0,C 180,E1 -11066.947,E2 -11066.947} C_VEL
LIN {X 0,Y 395.841,Z 684.643,A -85,B 0,C 180,E1 -11067.965,E2 -11067.965} C_VEL
LIN {X 0,Y 395.779,Z 685.494,A -85,B 0,C 180,E1 -11070,E2 -11070} C_VEL
LIN {X 0,Y 395.796,Z 685.303,A -85,B 0,C 180,E1 -11071.017,E2 -11071.017} C_VEL
LIN {X 0,Y 395.842,Z 684.717,A -85,B 0,C 180,E1 -11072.035,E2 -11072.035} C_VEL
LIN {X 0,Y 395.845,Z 683.751,A -85,B 0,C 180,E1 -11073.053,E2 -11073.053} C_VEL
LIN {X 0,Y 395.879,Z 682.388,A -85,B 0,C 180,E1 -11074.072,E2 -11074.072} C_VEL
LIN {X 0,Y 396.119,Z 679.516,A -85,B 0,C 180,E1 -11075.6,E2 -11075.6} C_VEL
LIN {X 0,Y 396.308,Z 675.618,A -85,B 0,C 180,E1 -11077.131,E2 -11077.131} C_VEL
LIN {X 0,Y 396.684,Z 670.565,A -85,B 0,C 180,E1 -11078.661,E2 -11078.661} C_VEL
LIN {X 0,Y 397.245,Z 664.192,A -85,B 0,C 180,E1 -11080.19,E2 -11080.19} C_VEL
LIN {X 0,Y 397.929,Z 656.276,A -85,B 0,C 180,E1 -11081.719,E2 -11081.719} C_VEL
LIN {X 0,Y 398.703,Z 648.183,A -85,B 0,C 180,E1 -11082.988,E2 -11082.988} C_VEL
LIN {X 0,Y 399.544,Z 638.238,A -85,B 0,C 180,E1 -11084.256,E2 -11084.256} C_VEL
LIN {X 0,Y 400.328,Z 627.061,A -85,B 0,C 180,E1 -11085.398,E2 -11085.398} C_VEL
LIN {X 0,Y 401.072,Z 616.111,A -85,B 0,C 180,E1 -11086.282,E2 -11086.282} C_VEL
LIN {X 0,Y 401.79,Z 604.999,A -85,B 0,C 180,E1 -11086.971,E2 -11086.971} C_VEL
LIN {X 0,Y 402.356,Z 591.787,A -85,B 0,C 180,E1 -11087.569,E2 -11087.569} C_VEL
LIN {X 0,Y 402.719,Z 580.126,A -85,B 0,C 180,E1 -11087.914,E2 -11087.914} C_VEL
LIN {X 0,Y 403.718,Z 493.223,A -85,B 0,C 180,E1 -11089.489,E2 -11089.489} C_VEL
LIN {X 0,Y 399.981,Z 471.88,A -85,B 0,C 180,E1 -11090.088,E2 -11090.088} C_VEL
LIN {X 0,Y 400.643,Z 454.743,A -85,B 0,C 180,E1 -11092.974,E2 -11092.974} C_VEL
LIN {X 0,Y 401.209,Z 444.036,A -85,B 0,C 180,E1 -11094.861,E2 -11094.861} C_VEL
LIN {X 0,Y 399.224,Z 433.237,A -85,B 0,C 180,E1 -11096.973,E2 -11096.973} C_VEL
LIN {X 0,Y 397.117,Z 424.02,A -85,B 0,C 180,E1 -11098.833,E2 -11098.833} C_VEL
LIN {X 0,Y 397.081,Z 424.027,A -85,B 0,C 180,E1 -11102.072,E2 -11102.072} C_VEL
LIN {X 0,Y 397.121,Z 424.021,A -85,B 0,C 180,E1 -11105.503,E2 -11105.503} C_VEL
LIN {X 0,Y 397.13,Z 424.018,A -85,B 0,C 180,E1 -11108.861,E2 -11108.861} C_VEL
LIN {X 0,Y 397.071,Z 424.024,A -85,B 0,C 180,E1 -11112.267,E2 -11112.267} C_VEL
LIN {X 0,Y 397.092,Z 424.022,A -85,B 0,C 180,E1 -11115.068,E2 -11115.068} C_VEL
LIN {X 0,Y 397.07,Z 424.016,A -85,B 0,C 180,E1 -11118.021,E2 -11118.021} C_VEL
LIN {X 0,Y 397.133,Z 424.017,A -85,B 0,C 180,E1 -11121.138,E2 -11121.138} C_VEL
LIN {X 0,Y 397.121,Z 424.008,A -85,B 0,C 180,E1 -11124.497,E2 -11124.497} C_VEL
LIN {X 0,Y 397.081,Z 424.022,A -85,B 0,C 180,E1 -11127.928,E2 -11127.928} C_VEL
LIN {X 0,Y 397.115,Z 424.019,A -85,B 0,C 180,E1 -11131.456,E2 -11131.456} C_VEL
LIN {X 0,Y 397.156,Z 424.142,A -85,B 0,C 180,E1 -11131.846,E2 -11131.846} C_VEL
LIN {X 0,Y 400.339,Z 439.717,A -85,B 0,C 180,E1 -11134.804,E2 -11134.804} C_VEL
LIN {X 0,Y 400.773,Z 443.646,A -85,B 0,C 180,E1 -11135.527,E2 -11135.527} C_VEL
LIN {X 0,Y 399.953,Z 459.72,A -85,B 0,C 180,E1 -11138.345,E2 -11138.345} C_VEL
LIN {X 0,Y 399.43,Z 472.382,A -85,B 0,C 180,E1 -11140.55,E2 -11140.55} C_VEL
LIN {X 0,Y 402.582,Z 494.269,A -85,B 0,C 180,E1 -11141.181,E2 -11141.181} C_VEL
LIN {X 0,Y 400.831,Z 583.435,A -85,B 0,C 180,E1 -11143.151,E2 -11143.151} C_VEL
LIN {X 0,Y 400.38,Z 597.558,A -85,B 0,C 180,E1 -11143.689,E2 -11143.689} C_VEL
LIN {X 0,Y 399.867,Z 609.24,A -85,B 0,C 180,E1 -11144.322,E2 -11144.322} C_VEL
LIN {X 0,Y 399.203,Z 621.681,A -85,B 0,C 180,E1 -11145.21,E2 -11145.21} C_VEL
LIN {X 0,Y 398.744,Z 631.494,A -85,B 0,C 180,E1 -11146.092,E2 -11146.092} C_VEL
LIN {X 0,Y 398.125,Z 641.984,A -85,B 0,C 180,E1 -11147.252,E2 -11147.252} C_VEL
LIN {X 0,Y 397.473,Z 651.384,A -85,B 0,C 180,E1 -11148.526,E2 -11148.526} C_VEL
LIN {X 0,Y 396.961,Z 659.133,A -85,B 0,C 180,E1 -11149.802,E2 -11149.802} C_VEL
LIN {X 0,Y 396.513,Z 666.676,A -85,B 0,C 180,E1 -11151.335,E2 -11151.335} C_VEL
LIN {X 0,Y 396.213,Z 672.723,A -85,B 0,C 180,E1 -11152.867,E2 -11152.867} C_VEL
LIN {X 0,Y 396.019,Z 677.471,A -85,B 0,C 180,E1 -11154.399,E2 -11154.399} C_VEL
LIN {X 0,Y 395.856,Z 681.049,A -85,B 0,C 180,E1 -11155.928,E2 -11155.928} C_VEL
LIN {X 0,Y 395.802,Z 682.815,A -85,B 0,C 180,E1 -11156.946,E2 -11156.946} C_VEL
LIN {X 0,Y 395.82,Z 684.149,A -85,B 0,C 180,E1 -11157.965,E2 -11157.965} C_VEL
LIN {X 0,Y 395.796,Z 685.06,A -85,B 0,C 180,E1 -11158.983,E2 -11158.983} C_VEL
LIN {X 0,Y 395.779,Z 685.498,A -85,B 0,C 180,E1 -11160,E2 -11160} C_VEL
LIN {X 0,Y 395.797,Z 685.527,A -85,B 0,C 180,E1 -11161.017,E2 -11161.017} C_VEL
LIN {X 0,Y 395.881,Z 685.138,A -85,B 0,C 180,E1 -11162.035,E2 -11162.035} C_VEL
LIN {X 0,Y 395.895,Z 684.281,A -85,B 0,C 180,E1 -11163.053,E2 -11163.053} C_VEL
LIN {X 0,Y 395.885,Z 683.014,A -85,B 0,C 180,E1 -11164.072,E2 -11164.072} C_VEL
LIN {X 0,Y 396.185,Z 680.252,A -85,B 0,C 180,E1 -11165.599,E2 -11165.599} C_VEL
LIN {X 0,Y 396.358,Z 676.424,A -85,B 0,C 180,E1 -11167.13,E2 -11167.13} C_VEL
LIN {X 0,Y 396.768,Z 671.392,A -85,B 0,C 180,E1 -11168.659,E2 -11168.659} C_VEL
LIN {X 0,Y 397.316,Z 664.985,A -85,B 0,C 180,E1 -11170.188,E2 -11170.188} C_VEL
LIN {X 0,Y 398.051,Z 657.053,A -85,B 0,C 180,E1 -11171.715,E2 -11171.715} C_VEL
LIN {X 0,Y 398.723,Z 648.93,A -85,B 0,C 180,E1 -11172.987,E2 -11172.987} C_VEL
LIN {X 0,Y 399.595,Z 638.989,A -85,B 0,C 180,E1 -11174.254,E2 -11174.254} C_VEL
LIN {X 0,Y 400.47,Z 627.949,A -85,B 0,C 180,E1 -11175.393,E2 -11175.393} C_VEL
LIN {X 0,Y 401.294,Z 615.469,A -85,B 0,C 180,E1 -11176.404,E2 -11176.404} C_VEL
LIN {X 0,Y 402.065,Z 603.3,A -85,B 0,C 180,E1 -11177.156,E2 -11177.156} C_VEL
LIN {X 0,Y 402.735,Z 589.588,A -85,B 0,C 180,E1 -11177.781,E2 -11177.781} C_VEL
LIN {X 0,Y 403.338,Z 574.312,A -85,B 0,C 180,E1 -11178.213,E2 -11178.213} C_VEL
LIN {X 0,Y 405.729,Z 498.225,A -85,B 0,C 180,E1 -11180.082,E2 -11180.082} C_VEL
LIN {X 0,Y 405.677,Z 493.053,A -85,B 0,C 180,E1 -11180.234,E2 -11180.234} C_VEL
LIN {X 0,Y 402.784,Z 478.316,A -85,B 0,C 180,E1 -11180.889,E2 -11180.889} C_VEL
LIN {X 0,Y 401.845,Z 474.1,A -85,B 0,C 180,E1 -11181.11,E2 -11181.11} C_VEL
LIN {X 0,Y 403.082,Z 455.094,A -85,B 0,C 180,E1 -11184.463,E2 -11184.463} C_VEL
LIN {X 0,Y 403.421,Z 449.034,A -85,B 0,C 180,E1 -11185.542,E2 -11185.542} C_VEL
LIN {X 0,Y 402.242,Z 441.692,A -85,B 0,C 180,E1 -11187.018,E2 -11187.018} C_VEL
LIN {X 0,Y 399.626,Z 431.657,A -85,B 0,C 180,E1 -11189.211,E2 -11189.211} C_VEL
LIN {X 0,Y 397.092,Z 424.026,A -85,B 0,C 180,E1 -11191.029,E2 -11191.029} C_VEL
LIN {X 0,Y 397.127,Z 424.019,A -85,B 0,C 180,E1 -11194.493,E2 -11194.493} C_VEL
LIN {X 0,Y 397.105,Z 424.018,A -85,B 0,C 180,E1 -11198.275,E2 -11198.275} C_VEL
LIN {X 0,Y 397.09,Z 424.022,A -85,B 0,C 180,E1 -11200.909,E2 -11200.909} C_VEL
LIN {X 0,Y 397.103,Z 424.02,A -85,B 0,C 180,E1 -11203.648,E2 -11203.648} C_VEL
LIN {X 0,Y 397.104,Z 424.021,A -85,B 0,C 180,E1 -11206.521,E2 -11206.521} C_VEL
LIN {X 0,Y 397.116,Z 424.017,A -85,B 0,C 180,E1 -11210.423,E2 -11210.423} C_VEL
LIN {X 0,Y 397.11,Z 424.017,A -85,B 0,C 180,E1 -11214.265,E2 -11214.265} C_VEL
LIN {X 0,Y 397.117,Z 424.019,A -85,B 0,C 180,E1 -11216.727,E2 -11216.727} C_VEL
LIN {X 0,Y 397.14,Z 424.119,A -85,B 0,C 180,E1 -11218.975,E2 -11218.975} C_VEL
LIN {X 0,Y 400.776,Z 441.352,A -85,B 0,C 180,E1 -11222.309,E2 -11222.309} C_VEL
LIN {X 0,Y 401.276,Z 446.016,A -85,B 0,C 180,E1 -11223.169,E2 -11223.169} C_VEL
LIN {X 0,Y 399.757,Z 467.818,A -85,B 0,C 180,E1 -11226.973,E2 -11226.973} C_VEL
LIN {X 0,Y 399.162,Z 477.192,A -85,B 0,C 180,E1 -11228.583,E2 -11228.583} C_VEL
LIN {X 0,Y 400.194,Z 485.95,A -85,B 0,C 180,E1 -11229.122,E2 -11229.122} C_VEL
LIN {X 0,Y 402.546,Z 502.19,A -85,B 0,C 180,E1 -11229.796,E2 -11229.796} C_VEL
LIN {X 0,Y 404.185,Z 522.48,A -85,B 0,C 180,E1 -11230.51,E2 -11230.51} C_VEL
LIN {X 0,Y 402.301,Z 577.859,A -85,B 0,C 180,E1 -11231.903,E2 -11231.903} C_VEL
LIN {X 0,Y 401.891,Z 604.817,A -85,B 0,C 180,E1 -11232.41,E2 -11232.41} C_VEL
LIN {X 0,Y 401.352,Z 618.466,A -85,B 0,C 180,E1 -11232.878,E2 -11232.878} C_VEL
LIN {X 0,Y 400.71,Z 630.748,A -85,B 0,C 180,E1 -11233.506,E2 -11233.506} C_VEL
LIN {X 0,Y 399.902,Z 642.504,A -85,B 0,C 180,E1 -11234.323,E2 -11234.323} C_VEL
LIN {X 0,Y 399.142,Z 653.797,A -85,B 0,C 180,E1 -11235.338,E2 -11235.338} C_VEL
LIN {X 0,Y 398.27,Z 664.327,A -85,B 0,C 180,E1 -11236.527,E2 -11236.527} C_VEL
LIN {X 0,Y 397.615,Z 673.071,A -85,B 0,C 180,E1 -11237.754,E2 -11237.754} C_VEL
LIN {X 0,Y 396.892,Z 681.927,A -85,B 0,C 180,E1 -11239.285,E2 -11239.285} C_VEL
LIN {X 0,Y 396.412,Z 689.025,A -85,B 0,C 180,E1 -11240.819,E2 -11240.819} C_VEL
LIN {X 0,Y 396.074,Z 694.674,A -85,B 0,C 180,E1 -11242.352,E2 -11242.352} C_VEL
LIN {X 0,Y 395.91,Z 699.142,A -85,B 0,C 180,E1 -11243.886,E2 -11243.886} C_VEL
LIN {X 0,Y 395.891,Z 701.562,A -85,B 0,C 180,E1 -11244.908,E2 -11244.908} C_VEL
LIN {X 0,Y 395.843,Z 703.467,A -85,B 0,C 180,E1 -11245.928,E2 -11245.928} C_VEL
LIN {X 0,Y 395.809,Z 704.893,A -85,B 0,C 180,E1 -11246.947,E2 -11246.947} C_VEL
LIN {X 0,Y 395.835,Z 705.889,A -85,B 0,C 180,E1 -11247.965,E2 -11247.965} C_VEL
LIN {X 0,Y 395.831,Z 706.58,A -85,B 0,C 180,E1 -11250,E2 -11250} C_VEL
LIN {X 0,Y 395.837,Z 706.357,A -85,B 0,C 180,E1 -11251.017,E2 -11251.017} C_VEL
LIN {X 0,Y 395.838,Z 705.74,A -85,B 0,C 180,E1 -11252.035,E2 -11252.035} C_VEL
LIN {X 0,Y 395.815,Z 704.729,A -85,B 0,C 180,E1 -11253.053,E2 -11253.053} C_VEL
LIN {X 0,Y 395.849,Z 703.296,A -85,B 0,C 180,E1 -11254.072,E2 -11254.072} C_VEL
LIN {X 0,Y 395.858,Z 700.312,A -85,B 0,C 180,E1 -11255.604,E2 -11255.604} C_VEL
LIN {X 0,Y 396.055,Z 696.263,A -85,B 0,C 180,E1 -11257.135,E2 -11257.135} C_VEL
LIN {X 0,Y 396.375,Z 690.015,A -85,B 0,C 180,E1 -11258.925,E2 -11258.925} C_VEL
LIN {X 0,Y 396.813,Z 683.197,A -85,B 0,C 180,E1 -11260.459,E2 -11260.459} C_VEL
LIN {X 0,Y 397.363,Z 676.22,A -85,B 0,C 180,E1 -11261.736,E2 -11261.736} C_VEL
LIN {X 0,Y 398.04,Z 667.785,A -85,B 0,C 180,E1 -11263.01,E2 -11263.01} C_VEL
LIN {X 0,Y 398.824,Z 657.34,A -85,B 0,C 180,E1 -11264.283,E2 -11264.283} C_VEL
LIN {X 0,Y 399.591,Z 646.984,A -85,B 0,C 180,E1 -11265.297,E2 -11265.297} C_VEL
LIN {X 0,Y 400.388,Z 635.565,A -85,B 0,C 180,E1 -11266.18,E2 -11266.18} C_VEL
LIN {X 0,Y 401.127,Z 623.703,A -85,B 0,C 180,E1 -11266.869,E2 -11266.869} C_VEL
LIN {X 0,Y 401.714,Z 610.888,A -85,B 0,C 180,E1 -11267.401,E2 -11267.401} C_VEL
LIN {X 0,Y 402.29,Z 598.082,A -85,B 0,C 180,E1 -11267.835,E2 -11267.835} C_VEL
LIN {X 0,Y 402.878,Z 582.425,A -85,B 0,C 180,E1 -11268.268,E2 -11268.268} C_VEL
LIN {X 0,Y 404.612,Z 520.9,A -85,B 0,C 180,E1 -11269.763,E2 -11269.763} C_VEL
LIN {X 0,Y 402.89,Z 501.15,A -85,B 0,C 180,E1 -11270.437,E2 -11270.437} C_VEL
LIN {X 0,Y 399.443,Z 479.901,A -85,B 0,C 180,E1 -11271.333,E2 -11271.333} C_VEL
LIN {X 0,Y 401.049,Z 460.93,A -85,B 0,C 180,E1 -11274.871,E2 -11274.871} C_VEL
LIN {X 0,Y 402.476,Z 447.092,A -85,B 0,C 180,E1 -11277.564,E2 -11277.564} C_VEL
LIN {X 0,Y 400.808,Z 438.042,A -85,B 0,C 180,E1 -11279.673,E2 -11279.673} C_VEL
LIN {X 0,Y 398.42,Z 428.633,A -85,B 0,C 180,E1 -11282.145,E2 -11282.145} C_VEL
LIN {X 0,Y 397.135,Z 424.018,A -85,B 0,C 180,E1 -11283.494,E2 -11283.494} C_VEL
LIN {X 0,Y 397.1,Z 424.023,A -85,B 0,C 180,E1 -11286.995,E2 -11286.995} C_VEL
LIN {X 0,Y 397.114,Z 424.02,A -85,B 0,C 180,E1 -11289.577,E2 -11289.577} C_VEL
LIN {X 0,Y 397.102,Z 424.02,A -85,B 0,C 180,E1 -11293.649,E2 -11293.649} C_VEL
LIN {X 0,Y 397.104,Z 424.02,A -85,B 0,C 180,E1 -11296.521,E2 -11296.521} C_VEL
LIN {X 0,Y 397.116,Z 424.018,A -85,B 0,C 180,E1 -11300.423,E2 -11300.423} C_VEL
LIN {X 0,Y 397.11,Z 424.018,A -85,B 0,C 180,E1 -11304.265,E2 -11304.265} C_VEL
LIN {X 0,Y 397.117,Z 424.02,A -85,B 0,C 180,E1 -11306.727,E2 -11306.727} C_VEL
LIN {X 0,Y 397.127,Z 424.017,A -85,B 0,C 180,E1 -11310.296,E2 -11310.296} C_VEL
LIN {X 0,Y 397.197,Z 424.011,A -85,B 0,C 180,E1 -11312.61,E2 -11312.61} C_VEL
LIN {X 0,Y 397.135,Z 424.02,A -85,B 0,C 180,E1 -11315.982,E2 -11315.982} C_VEL
LIN {X 0,Y 397.127,Z 424.071,A -85,B 0,C 180,E1 -11318.59,E2 -11318.59} C_VEL
LIN {X 0,Y 398.149,Z 426.933,A -85,B 0,C 180,E1 -11318.775,E2 -11318.775} C_VEL
LIN {X 0,Y 400.511,Z 431.132,A -85,B 0,C 180,E1 -11319.123,E2 -11319.123} C_VEL
LIN {X 0,Y 406.193,Z 443.243,A -85,B 0,C 180,E1 -11319.96,E2 -11319.96} C_VEL
LIN {X 0,Y 406.311,Z 446.244,A -85,B 0,C 180,E1 -11320.058,E2 -11320.058} C_VEL
LIN {X 0,Y 404.04,Z 509.8,A -85,B 0,C 180,E1 -11321.656,E2 -11321.656} C_VEL
LIN {X 0,Y 403.588,Z 528.687,A -85,B 0,C 180,E1 -11322.159,E2 -11322.159} C_VEL
LIN {X 0,Y 403.236,Z 540.236,A -85,B 0,C 180,E1 -11322.634,E2 -11322.634} C_VEL
LIN {X 0,Y 402.77,Z 551.557,A -85,B 0,C 180,E1 -11323.267,E2 -11323.267} C_VEL
LIN {X 0,Y 402.084,Z 562.939,A -85,B 0,C 180,E1 -11324.092,E2 -11324.092} C_VEL
LIN {X 0,Y 401.236,Z 574.519,A -85,B 0,C 180,E1 -11325.157,E2 -11325.157} C_VEL
LIN {X 0,Y 400.477,Z 584.45,A -85,B 0,C 180,E1 -11326.296,E2 -11326.296} C_VEL
LIN {X 0,Y 399.666,Z 593.39,A -85,B 0,C 180,E1 -11327.56,E2 -11327.56} C_VEL
LIN {X 0,Y 398.871,Z 602.075,A -85,B 0,C 180,E1 -11329.082,E2 -11329.082} C_VEL
LIN {X 0,Y 398.236,Z 607.946,A -85,B 0,C 180,E1 -11330.349,E2 -11330.349} C_VEL
LIN {X 0,Y 397.673,Z 613.66,A -85,B 0,C 180,E1 -11331.872,E2 -11331.872} C_VEL
LIN {X 0,Y 397.136,Z 618.127,A -85,B 0,C 180,E1 -11333.395,E2 -11333.395} C_VEL
LIN {X 0,Y 396.972,Z 621.432,A -85,B 0,C 180,E1 -11334.922,E2 -11334.922} C_VEL
LIN {X 0,Y 396.717,Z 623.054,A -85,B 0,C 180,E1 -11335.937,E2 -11335.937} C_VEL
LIN {X 0,Y 396.432,Z 624.26,A -85,B 0,C 180,E1 -11336.951,E2 -11336.951} C_VEL
LIN {X 0,Y 396.238,Z 625.046,A -85,B 0,C 180,E1 -11337.967,E2 -11337.967} C_VEL
LIN {X 0,Y 396.146,Z 625.363,A -85,B 0,C 180,E1 -11338.984,E2 -11338.984} C_VEL
LIN {X 0,Y 396.106,Z 625.257,A -85,B 0,C 180,E1 -11340,E2 -11340} C_VEL
LIN {X 0,Y 396.12,Z 624.741,A -85,B 0,C 180,E1 -11341.017,E2 -11341.017} C_VEL
LIN {X 0,Y 396.217,Z 623.793,A -85,B 0,C 180,E1 -11342.033,E2 -11342.033} C_VEL
LIN {X 0,Y 396.393,Z 622.386,A -85,B 0,C 180,E1 -11343.049,E2 -11343.049} C_VEL
LIN {X 0,Y 396.577,Z 619.479,A -85,B 0,C 180,E1 -11344.574,E2 -11344.574} C_VEL
LIN {X 0,Y 396.622,Z 615.514,A -85,B 0,C 180,E1 -11346.103,E2 -11346.103} C_VEL
LIN {X 0,Y 396.987,Z 609.394,A -85,B 0,C 180,E1 -11347.886,E2 -11347.886} C_VEL
LIN {X 0,Y 397.371,Z 602.631,A -85,B 0,C 180,E1 -11349.416,E2 -11349.416} C_VEL
LIN {X 0,Y 397.912,Z 594.202,A -85,B 0,C 180,E1 -11350.945,E2 -11350.945} C_VEL
LIN {X 0,Y 398.4,Z 585.592,A -85,B 0,C 180,E1 -11352.221,E2 -11352.221} C_VEL
LIN {X 0,Y 399.01,Z 576.188,A -85,B 0,C 180,E1 -11353.367,E2 -11353.367} C_VEL
LIN {X 0,Y 399.558,Z 565.761,A -85,B 0,C 180,E1 -11354.403,E2 -11354.403} C_VEL
LIN {X 0,Y 400.069,Z 553.095,A -85,B 0,C 180,E1 -11355.409,E2 -11355.409} C_VEL
LIN {X 0,Y 400.545,Z 540.322,A -85,B 0,C 180,E1 -11356.173,E2 -11356.173} C_VEL
LIN {X 0,Y 400.944,Z 527.065,A -85,B 0,C 180,E1 -11356.746,E2 -11356.746} C_VEL
LIN {X 0,Y 401.171,Z 513.114,A -85,B 0,C 180,E1 -11357.13,E2 -11357.13} C_VEL
LIN {X 0,Y 402.582,Z 440.801,A -85,B 0,C 180,E1 -11358.708,E2 -11358.708} C_VEL
LIN {X 0,Y 397.136,Z 424.023,A -85,B 0,C 180,E1 -11359.339,E2 -11359.339} C_VEL
LIN {X 0,Y 397.114,Z 424.016,A -85,B 0,C 180,E1 -11363.032,E2 -11363.032} C_VEL
LIN {X 0,Y 397.136,Z 424.013,A -85,B 0,C 180,E1 -11366.258,E2 -11366.258} C_VEL
LIN {X 0,Y 397.124,Z 424.012,A -85,B 0,C 180,E1 -11368.544,E2 -11368.544} C_VEL
LIN {X 0,Y 397.081,Z 424.013,A -85,B 0,C 180,E1 -11372.072,E2 -11372.072} C_VEL
LIN {X 0,Y 397.122,Z 424.014,A -85,B 0,C 180,E1 -11375.503,E2 -11375.503} C_VEL
LIN {X 0,Y 397.131,Z 424.014,A -85,B 0,C 180,E1 -11378.861,E2 -11378.861} C_VEL
LIN {X 0,Y 397.071,Z 424.022,A -85,B 0,C 180,E1 -11382.267,E2 -11382.267} C_VEL
LIN {X 0,Y 397.089,Z 424.013,A -85,B 0,C 180,E1 -11385.069,E2 -11385.069} C_VEL
LIN {X 0,Y 397.069,Z 424.023,A -85,B 0,C 180,E1 -11388.021,E2 -11388.021} C_VEL
LIN {X 0,Y 397.13,Z 424.018,A -85,B 0,C 180,E1 -11391.139,E2 -11391.139} C_VEL
LIN {X 0,Y 397.121,Z 424.02,A -85,B 0,C 180,E1 -11394.497,E2 -11394.497} C_VEL
LIN {X 0,Y 397.081,Z 424.023,A -85,B 0,C 180,E1 -11397.928,E2 -11397.928} C_VEL
LIN {X 0,Y 397.142,Z 424.107,A -85,B 0,C 180,E1 -11401.313,E2 -11401.313} C_VEL
LIN {X 0,Y 400.361,Z 438.868,A -85,B 0,C 180,E1 -11404.249,E2 -11404.249} C_VEL
LIN {X 0,Y 401.156,Z 443.452,A -85,B 0,C 180,E1 -11405.136,E2 -11405.136} C_VEL
LIN {X 0,Y 400.384,Z 460.305,A -85,B 0,C 180,E1 -11408.099,E2 -11408.099} C_VEL
LIN {X 0,Y 399.947,Z 471.873,A -85,B 0,C 180,E1 -11410.009,E2 -11410.009} C_VEL
LIN {X 0,Y 403.779,Z 493.79,A -85,B 0,C 180,E1 -11410.623,E2 -11410.623} C_VEL
LIN {X 0,Y 402.642,Z 578.815,A -85,B 0,C 180,E1 -11412.149,E2 -11412.149} C_VEL
LIN {X 0,Y 402.314,Z 591.8,A -85,B 0,C 180,E1 -11412.527,E2 -11412.527} C_VEL
LIN {X 0,Y 401.757,Z 604.396,A -85,B 0,C 180,E1 -11413.093,E2 -11413.093} C_VEL
LIN {X 0,Y 401.036,Z 616.54,A -85,B 0,C 180,E1 -11413.847,E2 -11413.847} C_VEL
LIN {X 0,Y 400.289,Z 627.406,A -85,B 0,C 180,E1 -11414.73,E2 -11414.73} C_VEL
LIN {X 0,Y 399.577,Z 638.514,A -85,B 0,C 180,E1 -11415.875,E2 -11415.875} C_VEL
LIN {X 0,Y 399.333,Z 641.398,A -85,B 0,C 180,E1 -11416.22,E2 -11416.22} C_VEL
LIN {X 0,Y 398.255,Z 645.851,A -85,B 0,C 180,E1 -11416.763,E2 -11416.763} C_VEL
LIN {X 0,Y 394.764,Z 652.724,A -85,B 0,C 180,E1 -11417.667,E2 -11417.667} C_VEL
LIN {X 0,Y 391.363,Z 659.072,A -85,B 0,C 180,E1 -11418.66,E2 -11418.66} C_VEL
LIN {X 0,Y 390.426,Z 662.574,A -85,B 0,C 180,E1 -11419.334,E2 -11419.334} C_VEL
LIN {X 0,Y 389.866,Z 668.415,A -85,B 0,C 180,E1 -11420.663,E2 -11420.663} C_VEL
LIN {X 0,Y 389.373,Z 673.941,A -85,B 0,C 180,E1 -11422.22,E2 -11422.22} C_VEL
LIN {X 0,Y 389.132,Z 678.274,A -85,B 0,C 180,E1 -11423.779,E2 -11423.779} C_VEL
LIN {X 0,Y 388.995,Z 680.554,A -85,B 0,C 180,E1 -11424.817,E2 -11424.817} C_VEL
LIN {X 0,Y 388.807,Z 682.417,A -85,B 0,C 180,E1 -11425.854,E2 -11425.854} C_VEL
LIN {X 0,Y 388.75,Z 683.838,A -85,B 0,C 180,E1 -11426.891,E2 -11426.891} C_VEL
LIN {X 0,Y 388.744,Z 684.833,A -85,B 0,C 180,E1 -11427.928,E2 -11427.928} C_VEL
LIN {X 0,Y 388.708,Z 685.682,A -85,B 0,C 180,E1 -11430,E2 -11430} C_VEL
LIN {X 0,Y 388.728,Z 685.491,A -85,B 0,C 180,E1 -11431.036,E2 -11431.036} C_VEL
LIN {X 0,Y 388.744,Z 684.905,A -85,B 0,C 180,E1 -11432.072,E2 -11432.072} C_VEL
LIN {X 0,Y 388.75,Z 683.94,A -85,B 0,C 180,E1 -11433.109,E2 -11433.109} C_VEL
LIN {X 0,Y 388.806,Z 682.576,A -85,B 0,C 180,E1 -11434.146,E2 -11434.146} C_VEL
LIN {X 0,Y 389.054,Z 679.703,A -85,B 0,C 180,E1 -11435.702,E2 -11435.702} C_VEL
LIN {X 0,Y 389.252,Z 675.805,A -85,B 0,C 180,E1 -11437.261,E2 -11437.261} C_VEL
LIN {X 0,Y 389.668,Z 670.75,A -85,B 0,C 180,E1 -11438.819,E2 -11438.819} C_VEL
LIN {X 0,Y 390.264,Z 664.376,A -85,B 0,C 180,E1 -11440.375,E2 -11440.375} C_VEL
LIN {X 0,Y 390.965,Z 656.457,A -85,B 0,C 180,E1 -11441.931,E2 -11441.931} C_VEL
LIN {X 0,Y 391.799,Z 648.362,A -85,B 0,C 180,E1 -11443.221,E2 -11443.221} C_VEL
LIN {X 0,Y 392.661,Z 638.413,A -85,B 0,C 180,E1 -11444.512,E2 -11444.512} C_VEL
LIN {X 0,Y 393.486,Z 627.231,A -85,B 0,C 180,E1 -11445.673,E2 -11445.673} C_VEL
LIN {X 0,Y 394.253,Z 616.273,A -85,B 0,C 180,E1 -11446.572,E2 -11446.572} C_VEL
LIN {X 0,Y 395.016,Z 605.147,A -85,B 0,C 180,E1 -11447.272,E2 -11447.272} C_VEL
LIN {X 0,Y 395.616,Z 591.914,A -85,B 0,C 180,E1 -11447.878,E2 -11447.878} C_VEL
LIN {X 0,Y 395.967,Z 580.212,A -85,B 0,C 180,E1 -11448.23,E2 -11448.23} C_VEL
LIN {X 0,Y 397.056,Z 494.329,A -85,B 0,C 180,E1 -11449.809,E2 -11449.809} C_VEL
LIN {X 0,Y 393.131,Z 471.857,A -85,B 0,C 180,E1 -11450.473,E2 -11450.473} C_VEL
LIN {X 0,Y 393.784,Z 456.286,A -85,B 0,C 180,E1 -11453.119,E2 -11453.119} C_VEL
LIN {X 0,Y 394.314,Z 445.153,A -85,B 0,C 180,E1 -11455.098,E2 -11455.098} C_VEL
LIN {X 0,Y 392.308,Z 434.695,A -85,B 0,C 180,E1 -11457.182,E2 -11457.182} C_VEL
LIN {X 0,Y 390.086,Z 424.897,A -85,B 0,C 180,E1 -11459.181,E2 -11459.181} C_VEL
LIN {X 0,Y 390.045,Z 424.901,A -85,B 0,C 180,E1 -11462.721,E2 -11462.721} C_VEL
LIN {X 0,Y 390.058,Z 424.902,A -85,B 0,C 180,E1 -11465.825,E2 -11465.825} C_VEL
LIN {X 0,Y 390.071,Z 424.897,A -85,B 0,C 180,E1 -11469.218,E2 -11469.218} C_VEL
LIN {X 0,Y 390.045,Z 424.899,A -85,B 0,C 180,E1 -11472.374,E2 -11472.374} C_VEL
LIN {X 0,Y 390.049,Z 424.903,A -85,B 0,C 180,E1 -11475.355,E2 -11475.355} C_VEL
LIN {X 0,Y 390.035,Z 424.892,A -85,B 0,C 180,E1 -11478.187,E2 -11478.187} C_VEL
LIN {X 0,Y 390.093,Z 424.897,A -85,B 0,C 180,E1 -11480.908,E2 -11480.908} C_VEL
LIN {X 0,Y 390.087,Z 424.888,A -85,B 0,C 180,E1 -11484.793,E2 -11484.793} C_VEL
LIN {X 0,Y 390.026,Z 424.904,A -85,B 0,C 180,E1 -11488.496,E2 -11488.496} C_VEL
LIN {X 0,Y 390.116,Z 425.03,A -85,B 0,C 180,E1 -11491.613,E2 -11491.613} C_VEL
LIN {X 0,Y 393.322,Z 440.589,A -85,B 0,C 180,E1 -11494.606,E2 -11494.606} C_VEL
LIN {X 0,Y 393.81,Z 445.58,A -85,B 0,C 180,E1 -11495.527,E2 -11495.527} C_VEL
LIN {X 0,Y 392.876,Z 464.215,A -85,B 0,C 180,E1 -11498.817,E2 -11498.817} C_VEL
LIN {X 0,Y 392.507,Z 472.607,A -85,B 0,C 180,E1 -11500.288,E2 -11500.288} C_VEL
LIN {X 0,Y 395.684,Z 494.952,A -85,B 0,C 180,E1 -11500.942,E2 -11500.942} C_VEL
LIN {X 0,Y 393.893,Z 583.347,A -85,B 0,C 180,E1 -11502.945,E2 -11502.945} C_VEL
LIN {X 0,Y 393.416,Z 596.768,A -85,B 0,C 180,E1 -11503.458,E2 -11503.458} C_VEL
LIN {X 0,Y 392.873,Z 609.713,A -85,B 0,C 180,E1 -11504.169,E2 -11504.169} C_VEL
LIN {X 0,Y 392.192,Z 622.086,A -85,B 0,C 180,E1 -11505.072,E2 -11505.072} C_VEL
LIN {X 0,Y 391.67,Z 632.93,A -85,B 0,C 180,E1 -11506.081,E2 -11506.081} C_VEL
LIN {X 0,Y 390.981,Z 643.336,A -85,B 0,C 180,E1 -11507.279,E2 -11507.279} C_VEL
LIN {X 0,Y 390.328,Z 652.555,A -85,B 0,C 180,E1 -11508.576,E2 -11508.576} C_VEL
LIN {X 0,Y 389.774,Z 661.453,A -85,B 0,C 180,E1 -11510.137,E2 -11510.137} C_VEL
LIN {X 0,Y 389.312,Z 668.628,A -85,B 0,C 180,E1 -11511.696,E2 -11511.696} C_VEL
LIN {X 0,Y 389.01,Z 675.195,A -85,B 0,C 180,E1 -11513.543,E2 -11513.543} C_VEL
LIN {X 0,Y 388.859,Z 679.946,A -85,B 0,C 180,E1 -11515.335,E2 -11515.335} C_VEL
LIN {X 0,Y 388.707,Z 682.867,A -85,B 0,C 180,E1 -11516.891,E2 -11516.891} C_VEL
LIN {X 0,Y 388.719,Z 684.235,A -85,B 0,C 180,E1 -11517.928,E2 -11517.928} C_VEL
LIN {X 0,Y 388.709,Z 685.195,A -85,B 0,C 180,E1 -11518.964,E2 -11518.964} C_VEL
LIN {X 0,Y 388.708,Z 685.684,A -85,B 0,C 180,E1 -11520,E2 -11520} C_VEL
LIN {X 0,Y 388.729,Z 685.745,A -85,B 0,C 180,E1 -11521.036,E2 -11521.036} C_VEL
LIN {X 0,Y 388.798,Z 685.396,A -85,B 0,C 180,E1 -11522.072,E2 -11522.072} C_VEL
LIN {X 0,Y 388.802,Z 684.582,A -85,B 0,C 180,E1 -11523.109,E2 -11523.109} C_VEL
LIN {X 0,Y 388.811,Z 683.338,A -85,B 0,C 180,E1 -11524.146,E2 -11524.146} C_VEL
LIN {X 0,Y 389.142,Z 680.621,A -85,B 0,C 180,E1 -11525.701,E2 -11525.701} C_VEL
LIN {X 0,Y 389.316,Z 676.846,A -85,B 0,C 180,E1 -11527.26,E2 -11527.26} C_VEL
LIN {X 0,Y 389.775,Z 671.906,A -85,B 0,C 180,E1 -11528.816,E2 -11528.816} C_VEL
LIN {X 0,Y 390.351,Z 665.605,A -85,B 0,C 180,E1 -11530.372,E2 -11530.372} C_VEL
LIN {X 0,Y 391.136,Z 657.734,A -85,B 0,C 180,E1 -11531.925,E2 -11531.925} C_VEL
LIN {X 0,Y 391.852,Z 649.705,A -85,B 0,C 180,E1 -11533.219,E2 -11533.219} C_VEL
LIN {X 0,Y 392.792,Z 639.851,A -85,B 0,C 180,E1 -11534.507,E2 -11534.507} C_VEL
LIN {X 0,Y 393.713,Z 629.045,A -85,B 0,C 180,E1 -11535.664,E2 -11535.664} C_VEL
LIN {X 0,Y 394.6,Z 616.895,A -85,B 0,C 180,E1 -11536.69,E2 -11536.69} C_VEL
LIN {X 0,Y 395.477,Z 604.115,A -85,B 0,C 180,E1 -11537.517,E2 -11537.517} C_VEL
LIN {X 0,Y 396.225,Z 589.836,A -85,B 0,C 180,E1 -11538.184,E2 -11538.184} C_VEL
LIN {X 0,Y 396.853,Z 574.664,A -85,B 0,C 180,E1 -11538.622,E2 -11538.622} C_VEL
LIN {X 0,Y 399.389,Z 502.652,A -85,B 0,C 180,E1 -11540.452,E2 -11540.452} C_VEL
LIN {X 0,Y 399.464,Z 494.402,A -85,B 0,C 180,E1 -11540.687,E2 -11540.687} C_VEL
LIN {X 0,Y 396.87,Z 480.794,A -85,B 0,C 180,E1 -11541.317,E2 -11541.317} C_VEL
LIN {X 0,Y 395.38,Z 474.448,A -85,B 0,C 180,E1 -11541.655,E2 -11541.655} C_VEL
LIN {X 0,Y 396.768,Z 454.906,A -85,B 0,C 180,E1 -11545.158,E2 -11545.158} C_VEL
LIN {X 0,Y 396.892,Z 450.381,A -85,B 0,C 180,E1 -11545.993,E2 -11545.993} C_VEL
LIN {X 0,Y 395.247,Z 441.791,A -85,B 0,C 180,E1 -11547.82,E2 -11547.82} C_VEL
LIN {X 0,Y 392.873,Z 433.361,A -85,B 0,C 180,E1 -11549.763,E2 -11549.763} C_VEL
LIN {X 0,Y 390.039,Z 424.905,A -85,B 0,C 180,E1 -11551.89,E2 -11551.89} C_VEL
LIN {X 0,Y 390.087,Z 424.895,A -85,B 0,C 180,E1 -11555.207,E2 -11555.207} C_VEL
LIN {X 0,Y 390.072,Z 424.896,A -85,B 0,C 180,E1 -11559.218,E2 -11559.218} C_VEL
LIN {X 0,Y 390.045,Z 424.9,A -85,B 0,C 180,E1 -11562.374,E2 -11562.374} C_VEL
LIN {X 0,Y 390.046,Z 424.898,A -85,B 0,C 180,E1 -11565.354,E2 -11565.354} C_VEL
LIN {X 0,Y 390.033,Z 424.902,A -85,B 0,C 180,E1 -11568.187,E2 -11568.187} C_VEL
LIN {X 0,Y 390.092,Z 424.891,A -85,B 0,C 180,E1 -11570.908,E2 -11570.908} C_VEL
LIN {X 0,Y 390.087,Z 424.892,A -85,B 0,C 180,E1 -11574.793,E2 -11574.793} C_VEL
LIN {X 0,Y 390.107,Z 425.044,A -85,B 0,C 180,E1 -11578.752,E2 -11578.752} C_VEL
LIN {X 0,Y 393.662,Z 441.794,A -85,B 0,C 180,E1 -11582.054,E2 -11582.054} C_VEL
LIN {X 0,Y 394.304,Z 445.559,A -85,B 0,C 180,E1 -11582.772,E2 -11582.772} C_VEL
LIN {X 0,Y 393.388,Z 459.041,A -85,B 0,C 180,E1 -11585.176,E2 -11585.176} C_VEL
LIN {X 0,Y 392.389,Z 473.567,A -85,B 0,C 180,E1 -11587.733,E2 -11587.733} C_VEL
LIN {X 0,Y 393.758,Z 485.333,A -85,B 0,C 180,E1 -11588.538,E2 -11588.538} C_VEL
LIN {X 0,Y 396.29,Z 502.815,A -85,B 0,C 180,E1 -11589.314,E2 -11589.314} C_VEL
LIN {X 0,Y 397.881,Z 523.046,A -85,B 0,C 180,E1 -11590.051,E2 -11590.051} C_VEL
LIN {X 0,Y 395.523,Z 590.499,A -85,B 0,C 180,E1 -11591.816,E2 -11591.816} C_VEL
LIN {X 0,Y 395.046,Z 606.958,A -85,B 0,C 180,E1 -11592.162,E2 -11592.162} C_VEL
LIN {X 0,Y 394.504,Z 619.819,A -85,B 0,C 180,E1 -11592.639,E2 -11592.639} C_VEL
LIN {X 0,Y 393.838,Z 631.585,A -85,B 0,C 180,E1 -11593.277,E2 -11593.277} C_VEL
LIN {X 0,Y 392.948,Z 643.907,A -85,B 0,C 180,E1 -11594.172,E2 -11594.172} C_VEL
LIN {X 0,Y 392.148,Z 654.891,A -85,B 0,C 180,E1 -11595.203,E2 -11595.203} C_VEL
LIN {X 0,Y 391.192,Z 665.726,A -85,B 0,C 180,E1 -11596.494,E2 -11596.494} C_VEL
LIN {X 0,Y 390.532,Z 674.512,A -85,B 0,C 180,E1 -11597.792,E2 -11597.792} C_VEL
LIN {X 0,Y 389.788,Z 683.049,A -85,B 0,C 180,E1 -11599.35,E2 -11599.35} C_VEL
LIN {X 0,Y 389.254,Z 690.896,A -85,B 0,C 180,E1 -11601.172,E2 -11601.172} C_VEL
LIN {X 0,Y 388.937,Z 696.271,A -85,B 0,C 180,E1 -11602.733,E2 -11602.733} C_VEL
LIN {X 0,Y 388.781,Z 700.13,A -85,B 0,C 180,E1 -11604.172,E2 -11604.172} C_VEL
LIN {X 0,Y 388.763,Z 703.38,A -85,B 0,C 180,E1 -11605.853,E2 -11605.853} C_VEL
LIN {X 0,Y 388.712,Z 704.779,A -85,B 0,C 180,E1 -11606.891,E2 -11606.891} C_VEL
LIN {X 0,Y 388.733,Z 705.742,A -85,B 0,C 180,E1 -11607.928,E2 -11607.928} C_VEL
LIN {X 0,Y 388.758,Z 706.391,A -85,B 0,C 180,E1 -11610,E2 -11610} C_VEL
LIN {X 0,Y 388.765,Z 706.169,A -85,B 0,C 180,E1 -11611.036,E2 -11611.036} C_VEL
LIN {X 0,Y 388.737,Z 705.55,A -85,B 0,C 180,E1 -11612.072,E2 -11612.072} C_VEL
LIN {X 0,Y 388.718,Z 704.54,A -85,B 0,C 180,E1 -11613.109,E2 -11613.109} C_VEL
LIN {X 0,Y 388.769,Z 703.107,A -85,B 0,C 180,E1 -11614.147,E2 -11614.147} C_VEL
LIN {X 0,Y 388.777,Z 699.834,A -85,B 0,C 180,E1 -11615.827,E2 -11615.827} C_VEL
LIN {X 0,Y 388.972,Z 696.073,A -85,B 0,C 180,E1 -11617.266,E2 -11617.266} C_VEL
LIN {X 0,Y 389.333,Z 689.826,A -85,B 0,C 180,E1 -11619.088,E2 -11619.088} C_VEL
LIN {X 0,Y 389.795,Z 683.009,A -85,B 0,C 180,E1 -11620.65,E2 -11620.65} C_VEL
LIN {X 0,Y 390.398,Z 676.033,A -85,B 0,C 180,E1 -11621.948,E2 -11621.948} C_VEL
LIN {X 0,Y 391.093,Z 667.6,A -85,B 0,C 180,E1 -11623.245,E2 -11623.245} C_VEL
LIN {X 0,Y 391.931,Z 657.158,A -85,B 0,C 180,E1 -11624.539,E2 -11624.539} C_VEL
LIN {X 0,Y 392.717,Z 646.806,A -85,B 0,C 180,E1 -11625.571,E2 -11625.571} C_VEL
LIN {X 0,Y 393.576,Z 635.393,A -85,B 0,C 180,E1 -11626.468,E2 -11626.468} C_VEL
LIN {X 0,Y 394.34,Z 623.541,A -85,B 0,C 180,E1 -11627.168,E2 -11627.168} C_VEL
LIN {X 0,Y 394.956,Z 610.743,A -85,B 0,C 180,E1 -11627.708,E2 -11627.708} C_VEL
LIN {X 0,Y 396.051,Z 591.551,A -85,B 0,C 180,E1 -11628.426,E2 -11628.426} C_VEL
LIN {X 0,Y 398.221,Z 521.698,A -85,B 0,C 180,E1 -11630.194,E2 -11630.194} C_VEL
LIN {X 0,Y 396.668,Z 502.825,A -85,B 0,C 180,E1 -11630.863,E2 -11630.863} C_VEL
LIN {X 0,Y 393.454,Z 482.554,A -85,B 0,C 180,E1 -11631.745,E2 -11631.745} C_VEL
LIN {X 0,Y 392.727,Z 478.647,A -85,B 0,C 180,E1 -11631.968,E2 -11631.968} C_VEL
LIN {X 0,Y 394.613,Z 459.793,A -85,B 0,C 180,E1 -11635.588,E2 -11635.588} C_VEL
LIN {X 0,Y 395.743,Z 448.879,A -85,B 0,C 180,E1 -11637.786,E2 -11637.786} C_VEL
LIN {X 0,Y 394.527,Z 441.801,A -85,B 0,C 180,E1 -11639.47,E2 -11639.47} C_VEL
LIN {X 0,Y 391.995,Z 431.611,A -85,B 0,C 180,E1 -11642.207,E2 -11642.207} C_VEL
LIN {X 0,Y 390.079,Z 424.897,A -85,B 0,C 180,E1 -11644.265,E2 -11644.265} C_VEL
LIN {X 0,Y 390.043,Z 424.902,A -85,B 0,C 180,E1 -11647.78,E2 -11647.78} C_VEL
LIN {X 0,Y 390.057,Z 424.898,A -85,B 0,C 180,E1 -11650.821,E2 -11650.821} C_VEL
LIN {X 0,Y 390.056,Z 424.898,A -85,B 0,C 180,E1 -11653.886,E2 -11653.886} C_VEL
LIN {X 0,Y 390.059,Z 424.897,A -85,B 0,C 180,E1 -11656.79,E2 -11656.79} C_VEL
LIN {X 0,Y 390.058,Z 424.897,A -85,B 0,C 180,E1 -11659.561,E2 -11659.561} C_VEL
LIN {X 0,Y 390.046,Z 424.9,A -85,B 0,C 180,E1 -11662.449,E2 -11662.449} C_VEL
LIN {X 0,Y 390.07,Z 424.894,A -85,B 0,C 180,E1 -11665.975,E2 -11665.975} C_VEL
LIN {X 0,Y 390.049,Z 424.899,A -85,B 0,C 180,E1 -11669.869,E2 -11669.869} C_VEL
LIN {X 0,Y 390.116,Z 424.895,A -85,B 0,C 180,E1 -11673.232,E2 -11673.232} C_VEL
LIN {X 0,Y 390.109,Z 424.897,A -85,B 0,C 180,E1 -11676.75,E2 -11676.75} C_VEL
LIN {X 0,Y 390.044,Z 424.903,A -85,B 0,C 180,E1 -11677.909,E2 -11677.909} C_VEL
LIN {X 0,Y 391.2,Z 427.975,A -85,B 0,C 180,E1 -11678.149,E2 -11678.149} C_VEL
LIN {X 0,Y 392.243,Z 429.716,A -85,B 0,C 180,E1 -11678.308,E2 -11678.308} C_VEL
LIN {X 0,Y 398.509,Z 441.989,A -85,B 0,C 180,E1 -11679.284,E2 -11679.284} C_VEL
LIN {X 0,Y 400.179,Z 446.013,A -85,B 0,C 180,E1 -11679.552,E2 -11679.552} C_VEL
LIN {X 0,Y 397.183,Z 527.7,A -85,B 0,C 180,E1 -11681.695,E2 -11681.695} C_VEL
LIN {X 0,Y 396.748,Z 540.407,A -85,B 0,C 180,E1 -11682.208,E2 -11682.208} C_VEL
LIN {X 0,Y 396.285,Z 551.863,A -85,B 0,C 180,E1 -11682.852,E2 -11682.852} C_VEL
LIN {X 0,Y 395.598,Z 563.117,A -85,B 0,C 180,E1 -11683.668,E2 -11683.668} C_VEL
LIN {X 0,Y 394.768,Z 573.764,A -85,B 0,C 180,E1 -11684.644,E2 -11684.644} C_VEL
LIN {X 0,Y 393.887,Z 583.919,A -85,B 0,C 180,E1 -11685.798,E2 -11685.798} C_VEL
LIN {X 0,Y 393.036,Z 593.101,A -85,B 0,C 180,E1 -11687.084,E2 -11687.084} C_VEL
LIN {X 0,Y 392.183,Z 601.971,A -85,B 0,C 180,E1 -11688.631,E2 -11688.631} C_VEL
LIN {X 0,Y 391.343,Z 609.112,A -85,B 0,C 180,E1 -11690.177,E2 -11690.177} C_VEL
LIN {X 0,Y 390.737,Z 614.746,A -85,B 0,C 180,E1 -11691.727,E2 -11691.727} C_VEL
LIN {X 0,Y 390.176,Z 619.12,A -85,B 0,C 180,E1 -11693.276,E2 -11693.276} C_VEL
LIN {X 0,Y 389.957,Z 622.343,A -85,B 0,C 180,E1 -11694.83,E2 -11694.83} C_VEL
LIN {X 0,Y 389.694,Z 623.919,A -85,B 0,C 180,E1 -11695.863,E2 -11695.863} C_VEL
LIN {X 0,Y 389.397,Z 625.087,A -85,B 0,C 180,E1 -11696.896,E2 -11696.896} C_VEL
LIN {X 0,Y 389.191,Z 625.83,A -85,B 0,C 180,E1 -11697.93,E2 -11697.93} C_VEL
LIN {X 0,Y 389.091,Z 626.099,A -85,B 0,C 180,E1 -11698.965,E2 -11698.965} C_VEL
LIN {X 0,Y 389.05,Z 625.954,A -85,B 0,C 180,E1 -11700,E2 -11700} C_VEL
LIN {X 0,Y 389.066,Z 625.4,A -85,B 0,C 180,E1 -11701.035,E2 -11701.035} C_VEL
LIN {X 0,Y 389.172,Z 624.385,A -85,B 0,C 180,E1 -11702.07,E2 -11702.07} C_VEL
LIN {X 0,Y 389.323,Z 622.937,A -85,B 0,C 180,E1 -11703.104,E2 -11703.104} C_VEL
LIN {X 0,Y 389.529,Z 619.945,A -85,B 0,C 180,E1 -11704.657,E2 -11704.657} C_VEL
LIN {X 0,Y 389.582,Z 615.884,A -85,B 0,C 180,E1 -11706.214,E2 -11706.214} C_VEL
LIN {X 0,Y 389.946,Z 609.733,A -85,B 0,C 180,E1 -11708.003,E2 -11708.003} C_VEL
LIN {X 0,Y 390.348,Z 602.725,A -85,B 0,C 180,E1 -11709.587,E2 -11709.587} C_VEL
LIN {X 0,Y 390.915,Z 594.152,A -85,B 0,C 180,E1 -11711.144,E2 -11711.144} C_VEL
LIN {X 0,Y 391.507,Z 584.366,A -85,B 0,C 180,E1 -11712.572,E2 -11712.572} C_VEL
LIN {X 0,Y 392.178,Z 573.316,A -85,B 0,C 180,E1 -11713.868,E2 -11713.868} C_VEL
LIN {X 0,Y 392.797,Z 561.818,A -85,B 0,C 180,E1 -11714.943,E2 -11714.943} C_VEL
LIN {X 0,Y 393.229,Z 550.018,A -85,B 0,C 180,E1 -11715.817,E2 -11715.817} C_VEL
LIN {X 0,Y 393.742,Z 537.415,A -85,B 0,C 180,E1 -11716.527,E2 -11716.527} C_VEL
LIN {X 0,Y 394.093,Z 524.334,A -85,B 0,C 180,E1 -11717.046,E2 -11717.046} C_VEL
LIN {X 0,Y 394.449,Z 503.081,A -85,B 0,C 180,E1 -11717.565,E2 -11717.565} C_VEL
LIN {X 0,Y 395.622,Z 441.383,A -85,B 0,C 180,E1 -11718.965,E2 -11718.965} C_VEL
LIN {X 0,Y 390.117,Z 424.898,A -85,B 0,C 180,E1 -11719.574,E2 -11719.574} C_VEL
LIN {X 0,Y 390.068,Z 424.892,A -85,B 0,C 180,E1 -11723.352,E2 -11723.352} C_VEL
LIN {X 0,Y 390.115,Z 424.889,A -85,B 0,C 180,E1 -11726.768,E2 -11726.768} C_VEL
LIN {X 0,Y 390.042,Z 424.897,A -85,B 0,C 180,E1 -11730.3,E2 -11730.3} C_VEL
LIN {X 0,Y 390.07,Z 424.876,A -85,B 0,C 180,E1 -11734.025,E2 -11734.025} C_VEL
LIN {X 0,Y 390.045,Z 424.9,A -85,B 0,C 180,E1 -11737.551,E2 -11737.551} C_VEL
LIN {X 0,Y 390.059,Z 424.886,A -85,B 0,C 180,E1 -11740.821,E2 -11740.821} C_VEL
LIN {X 0,Y 390.057,Z 424.898,A -85,B 0,C 180,E1 -11743.886,E2 -11743.886} C_VEL
LIN {X 0,Y 390.06,Z 424.891,A -85,B 0,C 180,E1 -11746.79,E2 -11746.79} C_VEL
LIN {X 0,Y 390.059,Z 424.89,A -85,B 0,C 180,E1 -11749.561,E2 -11749.561} C_VEL
LIN {X 0,Y 390.045,Z 424.899,A -85,B 0,C 180,E1 -11752.449,E2 -11752.449} C_VEL
LIN {X 0,Y 390.07,Z 424.893,A -85,B 0,C 180,E1 -11755.975,E2 -11755.975} C_VEL
LIN {X 0,Y 390.039,Z 424.903,A -85,B 0,C 180,E1 -11759.7,E2 -11759.7} C_VEL
LIN {X 0,Y 390.117,Z 424.989,A -85,B 0,C 180,E1 -11760.988,E2 -11760.988} C_VEL
LIN {X 0,Y 393.463,Z 440.208,A -85,B 0,C 180,E1 -11764.048,E2 -11764.048} C_VEL
LIN {X 0,Y 394.283,Z 445.723,A -85,B 0,C 180,E1 -11765.121,E2 -11765.121} C_VEL
LIN {X 0,Y 393.453,Z 463.606,A -85,B 0,C 180,E1 -11768.256,E2 -11768.256} C_VEL
LIN {X 0,Y 393.098,Z 471.988,A -85,B 0,C 180,E1 -11769.646,E2 -11769.646} C_VEL
LIN {X 0,Y 397.052,Z 494.203,A -85,B 0,C 180,E1 -11770.287,E2 -11770.287} C_VEL
LIN {X 0,Y 396.213,Z 559.656,A -85,B 0,C 180,E1 -11771.481,E2 -11771.481} C_VEL
LIN {X 0,Y 395.824,Z 584.161,A -85,B 0,C 180,E1 -11771.964,E2 -11771.964} C_VEL
LIN {X 0,Y 395.344,Z 597.418,A -85,B 0,C 180,E1 -11772.443,E2 -11772.443} C_VEL
LIN {X 0,Y 394.684,Z 610.062,A -85,B 0,C 180,E1 -11773.114,E2 -11773.114} C_VEL
LIN {X 0,Y 393.892,Z 621.703,A -85,B 0,C 180,E1 -11773.945,E2 -11773.945} C_VEL
LIN {X 0,Y 393.076,Z 632.706,A -85,B 0,C 180,E1 -11774.961,E2 -11774.961} C_VEL
LIN {X 0,Y 392.312,Z 642.903,A -85,B 0,C 180,E1 -11776.137,E2 -11776.137} C_VEL
LIN {X 0,Y 391.439,Z 651.175,A -85,B 0,C 180,E1 -11777.294,E2 -11777.294} C_VEL
LIN {X 0,Y 390.765,Z 658.809,A -85,B 0,C 180,E1 -11778.589,E2 -11778.589} C_VEL
LIN {X 0,Y 390.426,Z 662.574,A -85,B 0,C 180,E1 -11779.334,E2 -11779.334} C_VEL
LIN {X 0,Y 389.524,Z 665.924,A -85,B 0,C 180,E1 -11780.036,E2 -11780.036} C_VEL
LIN {X 0,Y 386.284,Z 670.932,A -85,B 0,C 180,E1 -11781.205,E2 -11781.205} C_VEL
LIN {X 0,Y 383.044,Z 675.225,A -85,B 0,C 180,E1 -11782.449,E2 -11782.449} C_VEL
LIN {X 0,Y 382.158,Z 677.456,A -85,B 0,C 180,E1 -11783.259,E2 -11783.259} C_VEL
LIN {X 0,Y 381.92,Z 680.744,A -85,B 0,C 180,E1 -11784.721,E2 -11784.721} C_VEL
LIN {X 0,Y 381.737,Z 682.606,A -85,B 0,C 180,E1 -11785.777,E2 -11785.777} C_VEL
LIN {X 0,Y 381.657,Z 684.027,A -85,B 0,C 180,E1 -11786.833,E2 -11786.833} C_VEL
LIN {X 0,Y 381.643,Z 685.636,A -85,B 0,C 180,E1 -11788.945,E2 -11788.945} C_VEL
LIN {X 0,Y 381.622,Z 685.871,A -85,B 0,C 180,E1 -11790,E2 -11790} C_VEL
LIN {X 0,Y 381.643,Z 685.679,A -85,B 0,C 180,E1 -11791.055,E2 -11791.055} C_VEL
LIN {X 0,Y 381.656,Z 684.128,A -85,B 0,C 180,E1 -11793.167,E2 -11793.167} C_VEL
LIN {X 0,Y 381.736,Z 682.763,A -85,B 0,C 180,E1 -11794.223,E2 -11794.223} C_VEL
LIN {X 0,Y 381.989,Z 679.891,A -85,B 0,C 180,E1 -11795.808,E2 -11795.808} C_VEL
LIN {X 0,Y 382.208,Z 675.991,A -85,B 0,C 180,E1 -11797.395,E2 -11797.395} C_VEL
LIN {X 0,Y 382.64,Z 670.935,A -85,B 0,C 180,E1 -11798.982,E2 -11798.982} C_VEL
LIN {X 0,Y 383.271,Z 664.559,A -85,B 0,C 180,E1 -11800.566,E2 -11800.566} C_VEL
LIN {X 0,Y 384.017,Z 656.639,A -85,B 0,C 180,E1 -11802.15,E2 -11802.15} C_VEL
LIN {X 0,Y 384.895,Z 648.541,A -85,B 0,C 180,E1 -11803.463,E2 -11803.463} C_VEL
LIN {X 0,Y 385.806,Z 638.588,A -85,B 0,C 180,E1 -11804.775,E2 -11804.775} C_VEL
LIN {X 0,Y 386.646,Z 627.401,A -85,B 0,C 180,E1 -11805.958,E2 -11805.958} C_VEL
LIN {X 0,Y 387.454,Z 616.436,A -85,B 0,C 180,E1 -11806.871,E2 -11806.871} C_VEL
LIN {X 0,Y 388.252,Z 605.296,A -85,B 0,C 180,E1 -11807.582,E2 -11807.582} C_VEL
LIN {X 0,Y 388.883,Z 592.041,A -85,B 0,C 180,E1 -11808.199,E2 -11808.199} C_VEL
LIN {X 0,Y 389.23,Z 580.297,A -85,B 0,C 180,E1 -11808.557,E2 -11808.557} C_VEL
LIN {X 0,Y 390.409,Z 495.364,A -85,B 0,C 180,E1 -11810.142,E2 -11810.142} C_VEL
LIN {X 0,Y 386.313,Z 472.121,A -85,B 0,C 180,E1 -11810.83,E2 -11810.83} C_VEL
LIN {X 0,Y 386.983,Z 456.237,A -85,B 0,C 180,E1 -11813.55,E2 -11813.55} C_VEL
LIN {X 0,Y 387.484,Z 446.965,A -85,B 0,C 180,E1 -11815.202,E2 -11815.202} C_VEL
LIN {X 0,Y 385.733,Z 437.565,A -85,B 0,C 180,E1 -11817.097,E2 -11817.097} C_VEL
LIN {X 0,Y 383.04,Z 425.773,A -85,B 0,C 180,E1 -11819.545,E2 -11819.545} C_VEL
LIN {X 0,Y 383.006,Z 425.78,A -85,B 0,C 180,E1 -11823.401,E2 -11823.401} C_VEL
LIN {X 0,Y 383.034,Z 425.775,A -85,B 0,C 180,E1 -11826.164,E2 -11826.164} C_VEL
LIN {X 0,Y 383.011,Z 425.769,A -85,B 0,C 180,E1 -11829.958,E2 -11829.958} C_VEL
LIN {X 0,Y 383.007,Z 425.777,A -85,B 0,C 180,E1 -11832.779,E2 -11832.779} C_VEL
LIN {X 0,Y 383.002,Z 425.778,A -85,B 0,C 180,E1 -11835.79,E2 -11835.79} C_VEL
LIN {X 0,Y 382.991,Z 425.771,A -85,B 0,C 180,E1 -11838.796,E2 -11838.796} C_VEL
LIN {X 0,Y 383.002,Z 425.775,A -85,B 0,C 180,E1 -11842.096,E2 -11842.096} C_VEL
LIN {X 0,Y 383.02,Z 425.772,A -85,B 0,C 180,E1 -11845.332,E2 -11845.332} C_VEL
LIN {X 0,Y 382.984,Z 425.78,A -85,B 0,C 180,E1 -11849.081,E2 -11849.081} C_VEL
LIN {X 0,Y 383.045,Z 425.829,A -85,B 0,C 180,E1 -11851.358,E2 -11851.358} C_VEL
LIN {X 0,Y 386.289,Z 441.466,A -85,B 0,C 180,E1 -11854.399,E2 -11854.399} C_VEL
LIN {X 0,Y 386.878,Z 446.28,A -85,B 0,C 180,E1 -11855.303,E2 -11855.303} C_VEL
LIN {X 0,Y 386.031,Z 462.489,A -85,B 0,C 180,E1 -11858.202,E2 -11858.202} C_VEL
LIN {X 0,Y 385.581,Z 472.754,A -85,B 0,C 180,E1 -11860.016,E2 -11860.016} C_VEL
LIN {X 0,Y 388.785,Z 495.912,A -85,B 0,C 180,E1 -11860.708,E2 -11860.708} C_VEL
LIN {X 0,Y 386.928,Z 583.739,A -85,B 0,C 180,E1 -11862.765,E2 -11862.765} C_VEL
LIN {X 0,Y 386.443,Z 597.052,A -85,B 0,C 180,E1 -11863.287,E2 -11863.287} C_VEL
LIN {X 0,Y 385.881,Z 609.946,A -85,B 0,C 180,E1 -11864.01,E2 -11864.01} C_VEL
LIN {X 0,Y 385.182,Z 622.307,A -85,B 0,C 180,E1 -11864.93,E2 -11864.93} C_VEL
LIN {X 0,Y 384.671,Z 632.478,A -85,B 0,C 180,E1 -11865.884,E2 -11865.884} C_VEL
LIN {X 0,Y 383.932,Z 643.557,A -85,B 0,C 180,E1 -11867.176,E2 -11867.176} C_VEL
LIN {X 0,Y 383.323,Z 651.925,A -85,B 0,C 180,E1 -11868.365,E2 -11868.365} C_VEL
LIN {X 0,Y 382.818,Z 659.668,A -85,B 0,C 180,E1 -11869.689,E2 -11869.689} C_VEL
LIN {X 0,Y 382.33,Z 667.199,A -85,B 0,C 180,E1 -11871.277,E2 -11871.277} C_VEL
LIN {X 0,Y 382.062,Z 672.328,A -85,B 0,C 180,E1 -11872.602,E2 -11872.602} C_VEL
LIN {X 0,Y 381.825,Z 677.661,A -85,B 0,C 180,E1 -11874.336,E2 -11874.336} C_VEL
LIN {X 0,Y 381.715,Z 681.006,A -85,B 0,C 180,E1 -11875.776,E2 -11875.776} C_VEL
LIN {X 0,Y 381.616,Z 682.914,A -85,B 0,C 180,E1 -11876.833,E2 -11876.833} C_VEL
LIN {X 0,Y 381.619,Z 684.321,A -85,B 0,C 180,E1 -11877.889,E2 -11877.889} C_VEL
LIN {X 0,Y 381.61,Z 685.317,A -85,B 0,C 180,E1 -11878.945,E2 -11878.945} C_VEL
LIN {X 0,Y 381.621,Z 685.87,A -85,B 0,C 180,E1 -11880,E2 -11880} C_VEL
LIN {X 0,Y 381.645,Z 685.963,A -85,B 0,C 180,E1 -11881.055,E2 -11881.055} C_VEL
LIN {X 0,Y 381.702,Z 685.644,A -85,B 0,C 180,E1 -11882.11,E2 -11882.11} C_VEL
LIN {X 0,Y 381.71,Z 684.888,A -85,B 0,C 180,E1 -11883.166,E2 -11883.166} C_VEL
LIN {X 0,Y 381.741,Z 683.678,A -85,B 0,C 180,E1 -11884.223,E2 -11884.223} C_VEL
LIN {X 0,Y 382.1,Z 681.031,A -85,B 0,C 180,E1 -11885.806,E2 -11885.806} C_VEL
LIN {X 0,Y 382.287,Z 677.329,A -85,B 0,C 180,E1 -11887.394,E2 -11887.394} C_VEL
LIN {X 0,Y 382.795,Z 672.445,A -85,B 0,C 180,E1 -11888.978,E2 -11888.978} C_VEL
LIN {X 0,Y 383.398,Z 666.232,A -85,B 0,C 180,E1 -11890.563,E2 -11890.563} C_VEL
LIN {X 0,Y 384.229,Z 658.425,A -85,B 0,C 180,E1 -11892.143,E2 -11892.143} C_VEL
LIN {X 0,Y 384.989,Z 650.539,A -85,B 0,C 180,E1 -11893.459,E2 -11893.459} C_VEL
LIN {X 0,Y 385.995,Z 640.913,A -85,B 0,C 180,E1 -11894.768,E2 -11894.768} C_VEL
LIN {X 0,Y 386.985,Z 630.259,A -85,B 0,C 180,E1 -11895.943,E2 -11895.943} C_VEL
LIN {X 0,Y 387.927,Z 618.404,A -85,B 0,C 180,E1 -11896.986,E2 -11896.986} C_VEL
LIN {X 0,Y 388.919,Z 604.923,A -85,B 0,C 180,E1 -11897.891,E2 -11897.891} C_VEL
LIN {X 0,Y 389.757,Z 590.273,A -85,B 0,C 180,E1 -11898.599,E2 -11898.599} C_VEL
LIN {X 0,Y 390.419,Z 575.679,A -85,B 0,C 180,E1 -11899.043,E2 -11899.043} C_VEL
LIN {X 0,Y 393.225,Z 502.095,A -85,B 0,C 180,E1 -11900.976,E2 -11900.976} C_VEL
LIN {X 0,Y 393.253,Z 495.362,A -85,B 0,C 180,E1 -11901.183,E2 -11901.183} C_VEL
LIN {X 0,Y 390.372,Z 480.492,A -85,B 0,C 180,E1 -11901.918,E2 -11901.918} C_VEL
